KUKA KRL program: MyProgram_045().src

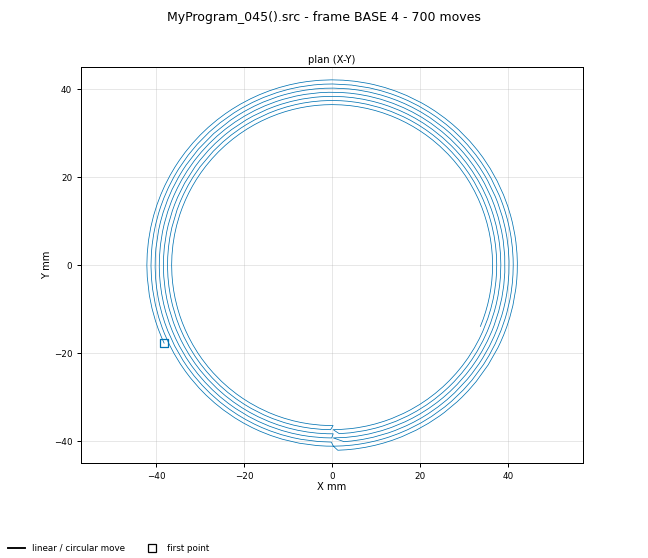
[picture p0: tool path of MyProgram_045().src in frame BASE 4, 700 of 700 moves have a stored position in this frame; points joined in program order, loops and branches not executed]
&ACCESS RVP
&REL 1
&PARAM TEMPLATE = C:\KRC\Roboter\Template\vorgabe
&PARAM EDITMASK = *
DEF MyProgram_045()
; ---- Setting reference (Base) ----
$BASE = BASE_DATA[4]

; --------------------------
; ---- Setting tool (TCP) ----
$TOOL = TOOL_DATA[3]
; --------------------------

$VEL.CP = VEL_APROX_PRINT
Startdeposition()
$VEL.CP = VEL_PRINT
LIN {X -38.1894,Y -17.7476,Z 64,A -162.0836,B 24.8594,C -2.7362,E1 24.8542,E2 -474.5644} C_DIS
LIN {X -38.8026,Y -16.3635,Z 64,A -164.3242,B 24.859,C -2.7399,E1 24.8517,E2 -472.3202} C_DIS
LIN {X -39.5429,Y -14.4833,Z 64,A -167.0478,B 24.8582,C -2.748,E1 24.849,E2 -469.6008} C_DIS
LIN {X -40.1481,Y -12.7091,Z 64,A -169.9379,B 24.8578,C -2.7517,E1 24.8465,E2 -466.703} C_DIS
LIN {X -40.9592,Y -9.7848,Z 64,A -173.7248,B 24.8561,C -2.7677,E1 24.8438,E2 -462.9324} C_DIS
LIN {X -41.5538,Y -6.8335,Z 64,A -178.6112,B 24.8557,C -2.7716,E1 24.8413,E2 -458.0262} C_DIS
LIN {X -42.0235,Y -2.7253,Z 64,A 175.6983,B 24.854,C -2.7884,E1 24.8399,E2 -452.3418} C_DIS
LIN {X -42.113,Y -0.0409,Z 64,A 172.223,B 24.8525,C -2.8017,E1 24.8399,E2 -448.8774} C_DIS
LIN {X -42.0286,Y 2.6491,Z 64,A 168.8043,B 24.8511,C -2.8158,E1 24.8403,E2 -445.4719} C_DIS
LIN {X -41.7458,Y 5.5413,Z 64,A 164.5763,B 24.85,C -2.8253,E1 24.8416,E2 -441.2413} C_DIS
LIN {X -41.2415,Y 8.5177,Z 64,A 160.7229,B 24.8484,C -2.8408,E1 24.8436,E2 -437.4022} C_DIS
LIN {X -40.5761,Y 11.2684,Z 64,A 157.2638,B 24.8467,C -2.8569,E1 24.846,E2 -433.9615} C_DIS
LIN {X -39.798,Y 13.7672,Z 64,A 152.9209,B 24.8464,C -2.8592,E1 24.8498,E2 -429.5994} C_DIS
LIN {X -38.9318,Y 16.0542,Z 64,A 150.3169,B 24.8445,C -2.8771,E1 24.8524,E2 -427.0234} C_DIS
LIN {X -38.035,Y 18.0757,Z 64,A 146.7752,B 24.8442,C -2.88,E1 24.8565,E2 -423.4695} C_DIS
LIN {X -36.8402,Y 20.4016,Z 64,A 143.3193,B 24.8429,C -2.8913,E1 24.8611,E2 -420.0222} C_DIS
LIN {X -35.7285,Y 22.2909,Z 64,A 140.4653,B 24.8419,C -2.901,E1 24.8652,E2 -417.1768} C_DIS
LIN {X -34.7653,Y 23.7657,Z 64,A 138.2662,B 24.8409,C -2.9098,E1 24.8686,E2 -414.9876} C_DIS
LIN {X -33.3953,Y 25.6547,Z 64,A 134.5117,B 24.8407,C -2.9116,E1 24.8749,E2 -411.2193} C_DIS
LIN {X -31.6682,Y 27.7586,Z 64,A 131.0357,B 24.8394,C -2.9235,E1 24.8811,E2 -407.7559} C_DIS
LIN {X -29.9941,Y 29.5595,Z 64,A 127.6294,B 24.8386,C -2.9308,E1 24.8877,E2 -404.3524} C_DIS
LIN {X -28.1817,Y 31.2924,Z 64,A 124.1921,B 24.8378,C -2.9383,E1 24.8947,E2 -400.9189} C_DIS
LIN {X -26.1567,Y 33.0036,Z 64,A 120.4268,B 24.8371,C -2.9441,E1 24.9028,E2 -397.1534} C_DIS
LIN {X -24.2784,Y 34.4092,Z 64,A 117.5539,B 24.836,C -2.9543,E1 24.9093,E2 -394.2946} C_DIS
LIN {X -22.7508,Y 35.4374,Z 64,A 115.1142,B 24.8354,C -2.9598,E1 24.915,E2 -391.8601} C_DIS
LIN {X -20.8416,Y 36.5931,Z 64,A 111.7463,B 24.8352,C -2.9611,E1 24.9231,E2 -388.4851} C_DIS
LIN {X -18.5524,Y 37.8048,Z 64,A 108.1834,B 24.8346,C -2.9662,E1 24.932,E2 -384.925} C_DIS
LIN {X -16.5365,Y 38.7294,Z 64,A 105.4902,B 24.8337,C -2.9746,E1 24.9388,E2 -382.2453} C_DIS
LIN {X -14.2871,Y 39.614,Z 64,A 101.6053,B 24.8341,C -2.9714,E1 24.949,E2 -378.3445} C_DIS
LIN {X -12.0392,Y 40.3542,Z 64,A 98.8345,B 24.833,C -2.9807,E1 24.9563,E2 -375.591} C_DIS
LIN {X -9.7408,Y 40.9696,Z 64,A 95.4963,B 24.8328,C -2.9825,E1 24.9654,E2 -372.2523} C_DIS
LIN {X -7.553,Y 41.4289,Z 64,A 92.4588,B 24.8325,C -2.9849,E1 24.9737,E2 -369.2174} C_DIS
LIN {X -5.5861,Y 41.7398,Z 64,A 89.5891,B 24.8325,C -2.9845,E1 24.9816,E2 -366.3443} C_DIS
LIN {X -2.9978,Y 42.0052,Z 64,A 86.1042,B 24.8323,C -2.9869,E1 24.9913,E2 -362.8635} C_DIS
LIN {X -0.1508,Y 42.1117,Z 64,A 82.6707,B 24.8315,C -2.994,E1 25.0008,E2 -359.4466} C_DIS
LIN {X 2.4941,Y 42.0383,Z 64,A 78.2258,B 24.8328,C -2.9825,E1 25.0133,E2 -354.9755} C_DIS
LIN {X 5.2133,Y 41.7881,Z 64,A 74.8519,B 24.8323,C -2.9867,E1 25.0226,E2 -351.6141} C_DIS
LIN {X 8.0189,Y 41.3412,Z 64,A 71.4094,B 24.8318,C -2.9915,E1 25.0321,E2 -348.1864} C_DIS
LIN {X 9.4728,Y 41.0326,Z 64,A 69.0763,B 24.8324,C -2.986,E1 25.0385,E2 -345.8434} C_DIS
LIN {X 12.0218,Y 40.3594,Z 64,A 65.3773,B 24.8329,C -2.982,E1 25.0484,E2 -342.141} C_DIS
LIN {X 14.4043,Y 39.5717,Z 64,A 62.0211,B 24.8331,C -2.9799,E1 25.0573,E2 -338.7867} C_DIS
LIN {X 16.9832,Y 38.5355,Z 64,A 57.7555,B 24.8344,C -2.9688,E1 25.0683,E2 -334.5046} C_DIS
LIN {X 20.3264,Y 36.882,Z 64,A 53.5076,B 24.8337,C -2.9749,E1 25.0787,E2 -330.2831} C_DIS
LIN {X 21.817,Y 36.0197,Z 64,A 50.7841,B 24.8347,C -2.9657,E1 25.0853,E2 -327.5461} C_DIS
LIN {X 23.4291,Y 34.9933,Z 64,A 48.2049,B 24.8351,C -2.9619,E1 25.0913,E2 -324.9666} C_DIS
LIN {X 25.6673,Y 33.3853,Z 64,A 44.808,B 24.8352,C -2.9611,E1 25.0989,E2 -321.5798} C_DIS
LIN {X 27.3862,Y 31.9908,Z 64,A 41.4445,B 24.8365,C -2.9499,E1 25.1061,E2 -318.2028} C_DIS
LIN {X 28.8143,Y 30.7107,Z 64,A 38.5792,B 24.8375,C -2.9406,E1 25.112,E2 -315.3271} C_DIS
LIN {X 31.3406,Y 28.1278,Z 64,A 34.5739,B 24.837,C -2.9449,E1 25.1197,E2 -311.3493} C_DIS
LIN {X 33.0583,Y 26.0874,Z 64,A 30.6147,B 24.8385,C -2.9312,E1 25.1268,E2 -307.3758} C_DIS
LIN {X 34.283,Y 24.4557,Z 64,A 27.4144,B 24.8401,C -2.9175,E1 25.132,E2 -304.1586} C_DIS
LIN {X 35.9427,Y 21.9439,Z 64,A 23.0552,B 24.8417,C -2.9027,E1 25.1385,E2 -299.7864} C_DIS
LIN {X 37.5319,Y 19.0985,Z 64,A 18.9072,B 24.8425,C -2.8956,E1 25.1439,E2 -295.6435} C_DIS
LIN {X 38.9801,Y 15.9362,Z 64,A 14.6589,B 24.843,C -2.8906,E1 25.1487,E2 -291.4064} C_DIS
LIN {X 39.9208,Y 13.4066,Z 64,A 10.6817,B 24.8447,C -2.8748,E1 25.1524,E2 -287.4142} C_DIS
LIN {X 40.5764,Y 11.2669,Z 64,A 8.1823,B 24.8447,C -2.8751,E1 25.1543,E2 -284.9298} C_DIS
LIN {X 40.9861,Y 9.6717,Z 64,A 5.0679,B 24.847,C -2.8535,E1 25.1564,E2 -281.7822} C_DIS
LIN {X 41.5467,Y 6.8764,Z 64,A 1.8676,B 24.847,C -2.8532,E1 25.158,E2 -278.6001} C_DIS
LIN {X 41.791,Y 5.1908,Z 64,A -0.8122,B 24.8485,C -2.8399,E1 25.1589,E2 -275.9045} C_DIS
LIN {X 42.0276,Y 2.6639,Z 64,A -3.7149,B 24.8486,C -2.8386,E1 25.1596,E2 -273.016} C_DIS
LIN {X 42.1073,Y 0.6196,Z 64,A -6.7943,B 24.8501,C -2.8248,E1 25.1598,E2 -269.9222} C_DIS
LIN {X 42.0818,Y -1.6027,Z 64,A -9.467,B 24.8505,C -2.8213,E1 25.1596,E2 -267.2572} C_DIS
LIN {X 41.9877,Y -3.2337,Z 64,A -11.5891,B 24.851,C -2.8161,E1 25.1592,E2 -265.1353} C_DIS
LIN {X 41.7761,Y -5.3062,Z 64,A -14.9089,B 24.8529,C -2.7988,E1 25.1581,E2 -261.7942} C_DIS
LIN {X 41.0947,Y -9.198,Z 64,A -20.5022,B 24.855,C -2.7783,E1 25.1551,E2 -256.1852} C_DIS
LIN {X 40.3709,Y -11.9829,Z 64,A -23.8222,B 24.8552,C -2.7765,E1 25.1526,E2 -252.8799} C_DIS
LIN {X 39.713,Y -14.0105,Z 64,A -26.748,B 24.8562,C -2.7672,E1 25.15,E2 -249.9486} C_DIS
LIN {X 39.0031,Y -15.8798,Z 64,A -29.3131,B 24.8567,C -2.7617,E1 25.1474,E2 -247.3848} C_DIS
LIN {X 38.2998,Y -17.5081,Z 64,A -31.798,B 24.8576,C -2.7533,E1 25.1446,E2 -244.8936} C_DIS
LIN {X 37.6614,Y -18.8428,Z 64,A -34.6547,B 24.8597,C -2.7331,E1 25.141,E2 -242.0043} C_DIS
LIN {X 35.4698,Y -22.7003,Z 64,A -40.7005,B 24.8615,C -2.7161,E1 25.1322,E2 -235.9491} C_DIS
LIN {X 32.7511,Y -26.4722,Z 64,A -46.2035,B 24.8617,C -2.7132,E1 25.123,E2 -230.4655} C_DIS
LIN {X 30.9506,Y -28.5566,Z 64,A -49.7785,B 24.8624,C -2.7067,E1 25.1164,E2 -226.8911} C_DIS
LIN {X 29.5084,Y -30.0446,Z 64,A -52.2115,B 24.8624,C -2.7064,E1 25.1116,E2 -224.4677} C_DIS
LIN {X 28.4019,Y -31.0925,Z 64,A -55.2369,B 24.8645,C -2.686,E1 25.1053,E2 -221.4062} C_DIS
LIN {X 25.523,Y -33.4965,Z 64,A -59.4397,B 24.8641,C -2.6897,E1 25.0963,E2 -217.2281} C_DIS
LIN {X 24.4241,Y -34.3055,Z 64,A -61.7378,B 24.8652,C -2.6788,E1 25.091,E2 -214.9122} C_DIS
LIN {X 21.9075,Y -35.9646,Z 64,A -65.825,B 24.866,C -2.6713,E1 25.0814,E2 -210.8205} C_DIS
LIN {X 19.1281,Y -37.5169,Z 64,A -70.6189,B 24.8675,C -2.6567,E1 25.0695,E2 -206.0057} C_DIS
LIN {X 15.8604,Y -39.0109,Z 64,A -74.9095,B 24.8672,C -2.6589,E1 25.0586,E2 -201.7306} C_DIS
LIN {X 13.743,Y -39.8058,Z 64,A -77.6711,B 24.8672,C -2.6598,E1 25.0514,E2 -198.977} C_DIS
LIN {X 11.7789,Y -40.4308,Z 64,A -80.9256,B 24.8682,C -2.6497,E1 25.0426,E2 -195.7043} C_DIS
LIN {X 9.793,Y -40.9572,Z 64,A -83.3321,B 24.8678,C -2.6529,E1 25.0362,E2 -193.3089} C_DIS
LIN {X 7.5807,Y -41.4241,Z 64,A -87.0071,B 24.869,C -2.6413,E1 25.026,E2 -189.6109} C_DIS
LIN {X 5.2253,Y -41.7866,Z 64,A -89.7045,B 24.8684,C -2.6473,E1 25.0186,E2 -186.9299} C_DIS
LIN {X 3.3156,Y -41.9811,Z 64,A -92.4426,B 24.8687,C -2.6441,E1 25.011,E2 -184.1858} C_DIS
LIN {X 1.2963,Y -42.0919,Z 64,A -95.1766,B 24.8688,C -2.6433,E1 25.0034,E2 -181.4508} C_DIS
LIN {X 1.2963,Y -42.0919,Z 64,A -95.1766,B 24.8688,C -2.6433,E1 25.0034,E2 -181.4508} C_DIS
Enddeposition()
LIN {X 0.2865,Y -41.1698,Z 64,A -95.4325,B 24.8656,C -2.6754,E1 25.0029,E2 -181.2711} C_DIS
Startdeposition()
$VEL.CP = VEL_PRINT
LIN {X 2.5086,Y -41.0971,Z 64,A -91.9997,B 24.865,C -2.6814,E1 25.0125,E2 -184.7172} C_DIS
LIN {X 4.5975,Y -40.9157,Z 64,A -89.3544,B 24.8652,C -2.679,E1 25.0198,E2 -187.3551} C_DIS
LIN {X 6.285,Y -40.6906,Z 64,A -86.9492,B 24.865,C -2.6811,E1 25.0264,E2 -189.7631} C_DIS
LIN {X 7.9842,Y -40.3918,Z 64,A -84.5187,B 24.8648,C -2.6835,E1 25.0331,E2 -192.1965} C_DIS
LIN {X 9.725,Y -40.0081,Z 64,A -81.9886,B 24.8645,C -2.6865,E1 25.04,E2 -194.7304} C_DIS
LIN {X 11.6702,Y -39.4844,Z 64,A -79.4566,B 24.8645,C -2.6854,E1 25.0468,E2 -197.2555} C_DIS
LIN {X 12.9333,Y -39.0895,Z 64,A -77.251,B 24.8638,C -2.6932,E1 25.0527,E2 -199.4754} C_DIS
LIN {X 15.0733,Y -38.3145,Z 64,A -74.3091,B 24.8638,C -2.6939,E1 25.0604,E2 -202.4126} C_DIS
LIN {X 17.1775,Y -37.4189,Z 64,A -70.4429,B 24.8621,C -2.7094,E1 25.0703,E2 -206.3061} C_DIS
LIN {X 20.208,Y -35.8732,Z 64,A -66.3938,B 24.8624,C -2.7063,E1 25.0802,E2 -210.3366} C_DIS
LIN {X 22.5789,Y -34.43,Z 64,A -61.6674,B 24.8603,C -2.7275,E1 25.0915,E2 -215.098} C_DIS
LIN {X 25.5833,Y -32.2598,Z 64,A -57.4368,B 24.8607,C -2.723,E1 25.1008,E2 -219.3026} C_DIS
LIN {X 27.1419,Y -30.9604,Z 64,A -54.1094,B 24.8592,C -2.7376,E1 25.1079,E2 -222.6515} C_DIS
LIN {X 29.8248,Y -28.3855,Z 64,A -48.7405,B 24.8576,C -2.7531,E1 25.1185,E2 -228.0344} C_DIS
LIN {X 31.799,Y -26.1552,Z 64,A -44.4279,B 24.8562,C -2.7665,E1 25.1263,E2 -232.359} C_DIS
LIN {X 34.4182,Y -22.5969,Z 64,A -39.348,B 24.8564,C -2.7649,E1 25.1344,E2 -237.4102} C_DIS
LIN {X 35.7205,Y -20.4761,Z 64,A -35.0283,B 24.8539,C -2.7892,E1 25.1406,E2 -241.7654} C_DIS
LIN {X 37.076,Y -17.9054,Z 64,A -31.2501,B 24.8531,C -2.7964,E1 25.1453,E2 -245.5404} C_DIS
LIN {X 38.4017,Y -14.8515,Z 64,A -26.6876,B 24.8518,C -2.809,E1 25.1502,E2 -250.1076} C_DIS
LIN {X 39.3357,Y -12.1622,Z 64,A -23.3798,B 24.8517,C -2.8098,E1 25.1531,E2 -253.3986} C_DIS
LIN {X 39.709,Y -10.8824,Z 64,A -21.0005,B 24.8501,C -2.8246,E1 25.1549,E2 -255.7991} C_DIS
LIN {X 40.3965,Y -7.9597,Z 64,A -17.258,B 24.8495,C -2.83,E1 25.1571,E2 -259.5328} C_DIS
LIN {X 40.6939,Y -6.2639,Z 64,A -14.7095,B 24.8485,C -2.8401,E1 25.1582,E2 -262.0904} C_DIS
LIN {X 40.9627,Y -4.1566,Z 64,A -11.8666,B 24.8477,C -2.8475,E1 25.1591,E2 -264.9337} C_DIS
LIN {X 41.1159,Y -2.1722,Z 64,A -9.0364,B 24.8466,C -2.8572,E1 25.1597,E2 -267.7702} C_DIS
LIN {X 41.1733,Y 0.0875,Z 64,A -6.0721,B 24.8459,C -2.864,E1 25.1597,E2 -270.7328} C_DIS
LIN {X 41.1424,Y 1.5996,Z 64,A -3.8198,B 24.8449,C -2.8731,E1 25.1596,E2 -272.9934} C_DIS
LIN {X 40.9794,Y 3.9883,Z 64,A -0.3005,B 24.8434,C -2.8867,E1 25.1587,E2 -276.5239} C_DIS
LIN {X 40.6864,Y 6.3124,Z 64,A 2.5108,B 24.8432,C -2.889,E1 25.1576,E2 -279.3241} C_DIS
LIN {X 40.3371,Y 8.2546,Z 64,A 5.8381,B 24.8412,C -2.9073,E1 25.1559,E2 -282.6755} C_DIS
LIN {X 39.8463,Y 10.3687,Z 64,A 8.2951,B 24.8412,C -2.9067,E1 25.1542,E2 -285.1167} C_DIS
LIN {X 39.3395,Y 12.1503,Z 64,A 10.9164,B 24.8403,C -2.915,E1 25.1521,E2 -287.7428} C_DIS
LIN {X 38.7443,Y 13.9319,Z 64,A 13.5664,B 24.8394,C -2.9232,E1 25.1497,E2 -290.3973} C_DIS
LIN {X 38.0364,Y 15.7633,Z 64,A 17.5379,B 24.8362,C -2.9521,E1 25.1454,E2 -294.4152} C_DIS
LIN {X 36.1894,Y 19.6355,Z 64,A 22.4347,B 24.8365,C -2.9499,E1 25.1392,E2 -299.2809} C_DIS
LIN {X 35.0453,Y 21.6121,Z 64,A 25.3732,B 24.836,C -2.9541,E1 25.135,E2 -302.2144} C_DIS
LIN {X 33.9192,Y 23.339,Z 64,A 28.1541,B 24.8354,C -2.9598,E1 25.1307,E2 -304.995} C_DIS
LIN {X 32.6665,Y 25.0626,Z 64,A 31.3409,B 24.8342,C -2.9706,E1 25.1253,E2 -308.192} C_DIS
LIN {X 30.7767,Y 27.3504,Z 64,A 35.0878,B 24.8338,C -2.9737,E1 25.1186,E2 -311.9291} C_DIS
LIN {X 29.3498,Y 28.876,Z 64,A 38.5961,B 24.832,C -2.9896,E1 25.1118,E2 -315.46} C_DIS
LIN {X 27.6483,Y 30.51,Z 64,A 41.6362,B 24.8317,C -2.9921,E1 25.1055,E2 -318.4938} C_DIS
LIN {X 25.9223,Y 31.9884,Z 64,A 44.7794,B 24.8311,C -2.9977,E1 25.0988,E2 -321.6382} C_DIS
LIN {X 23.7335,Y 33.6442,Z 64,A 48.6249,B 24.8303,C -3.0045,E1 25.0901,E2 -325.4862} C_DIS
LIN {X 22.074,Y 34.7558,Z 64,A 51.5102,B 24.8297,C -3.0105,E1 25.0833,E2 -328.3762} C_DIS
LIN {X 19.6272,Y 36.1939,Z 64,A 55.2494,B 24.8294,C -3.0126,E1 25.0742,E2 -332.1095} C_DIS
LIN {X 17.2767,Y 37.3731,Z 64,A 58.8016,B 24.8291,C -3.0153,E1 25.0653,E2 -335.6587} C_DIS
LIN {X 15.2195,Y 38.2569,Z 64,A 61.8902,B 24.8288,C -3.0181,E1 25.0574,E2 -338.7467} C_DIS
LIN {X 13.3989,Y 38.9323,Z 64,A 64.4426,B 24.8288,C -3.0181,E1 25.0507,E2 -341.2942} C_DIS
LIN {X 11.048,Y 39.6629,Z 64,A 68.5273,B 24.8274,C -3.0303,E1 25.0397,E2 -345.4006} C_DIS
LIN {X 8.5196,Y 40.2823,Z 64,A 72.2473,B 24.827,C -3.0334,E1 25.0295,E2 -349.1232} C_DIS
LIN {X 4.4101,Y 40.9362,Z 64,A 78.0835,B 24.8268,C -3.0354,E1 25.0134,E2 -354.9592} C_DIS
LIN {X 0.0841,Y 41.1734,Z 64,A 83.1585,B 24.8284,C -3.0216,E1 24.9993,E2 -359.9999} C_DIS
LIN {X -1.8757,Y 41.1298,Z 64,A 86.0866,B 24.8282,C -3.0235,E1 24.9911,E2 -362.9331} C_DIS
LIN {X -4.1334,Y 40.9648,Z 64,A 89.7492,B 24.8275,C -3.029,E1 24.9809,E2 -366.6105} C_DIS
LIN {X -7.42,Y 40.4984,Z 64,A 94.0771,B 24.8284,C -3.0219,E1 24.969,E2 -370.9255} C_DIS
LIN {X -9.8107,Y 39.9866,Z 64,A 97.8152,B 24.8282,C -3.0232,E1 24.9588,E2 -374.6717} C_DIS
LIN {X -12.5005,Y 39.2294,Z 64,A 101.6871,B 24.8287,C -3.0188,E1 24.9485,E2 -378.5396} C_DIS
LIN {X -15.6079,Y 38.1002,Z 64,A 105.9096,B 24.8299,C -3.008,E1 24.9375,E2 -382.7452} C_DIS
LIN {X -18.1335,Y 36.9647,Z 64,A 110.0885,B 24.8301,C -3.0062,E1 24.9269,E2 -386.9305} C_DIS
LIN {X -20.4211,Y 35.7522,Z 64,A 113.368,B 24.8313,C -2.9962,E1 24.9189,E2 -390.1954} C_DIS
LIN {X -22.2692,Y 34.6311,Z 64,A 116.6839,B 24.8315,C -2.9944,E1 24.9111,E2 -393.5176} C_DIS
LIN {X -25.4707,Y 32.3492,Z 64,A 122.5841,B 24.8321,C -2.9884,E1 24.8979,E2 -399.4246} C_DIS
LIN {X -27.954,Y 30.2292,Z 64,A 127.0418,B 24.8334,C -2.9773,E1 24.8886,E2 -403.8734} C_DIS
LIN {X -30.6733,Y 27.4659,Z 64,A 131.8749,B 24.8356,C -2.9577,E1 24.8794,E2 -408.6808} C_DIS
LIN {X -32.7326,Y 24.976,Z 64,A 137.3602,B 24.8356,C -2.9575,E1 24.8699,E2 -414.1913} C_DIS
LIN {X -34.9355,Y 21.7886,Z 64,A 141.9022,B 24.8383,C -2.9332,E1 24.8629,E2 -418.6978} C_DIS
LIN {X -36.0094,Y 19.964,Z 64,A 144.704,B 24.8394,C -2.9232,E1 24.8591,E2 -421.4905} C_DIS
LIN {X -37.206,Y 17.6331,Z 64,A 149.0173,B 24.8398,C -2.9201,E1 24.8537,E2 -425.8195} C_DIS
LIN {X -38.2384,Y 15.2655,Z 64,A 152.1055,B 24.8416,C -2.9038,E1 24.8505,E2 -428.886} C_DIS
LIN {X -38.9655,Y 13.3009,Z 64,A 154.8405,B 24.8427,C -2.8931,E1 24.8479,E2 -431.6108} C_DIS
LIN {X -39.4625,Y 11.7441,Z 64,A 157.4607,B 24.8431,C -2.8899,E1 24.8458,E2 -434.2385} C_DIS
LIN {X -40.1258,Y 9.226,Z 64,A 160.9334,B 24.8445,C -2.8771,E1 24.8434,E2 -437.7007} C_DIS
LIN {X -40.5485,Y 7.1441,Z 64,A 164.202,B 24.8451,C -2.8712,E1 24.8417,E2 -440.9748} C_DIS
LIN {X -40.908,Y 4.6637,Z 64,A 167.3897,B 24.8466,C -2.8571,E1 24.8406,E2 -444.1476} C_DIS
LIN {X -41.0794,Y 2.777,Z 64,A 170.5921,B 24.8469,C -2.8549,E1 24.8399,E2 -447.3641} C_DIS
LIN {X -41.1735,Y -0.1582,Z 64,A 174.2183,B 24.8488,C -2.8371,E1 24.8399,E2 -450.9696} C_DIS
LIN {X -41.0704,Y -2.9085,Z 64,A 178.4713,B 24.8496,C -2.8298,E1 24.8404,E2 -455.2307} C_DIS
LIN {X -40.8091,Y -5.4637,Z 64,A -177.2907,B 24.85,C -2.8261,E1 24.842,E2 -459.4852} C_DIS
LIN {X -40.1744,Y -9.0147,Z 64,A -172.6624,B 24.852,C -2.8066,E1 24.8446,E2 -464.0939} C_DIS
LIN {X -39.3951,Y -11.968,Z 64,A -168.8506,B 24.8539,C -2.7891,E1 24.8475,E2 -467.8861} C_DIS
LIN {X -38.6067,Y -14.3098,Z 64,A -165.727,B 24.8553,C -2.7757,E1 24.8503,E2 -470.9953} C_DIS
LIN {X -38.0815,Y -15.6538,Z 64,A -163.3316,B 24.8554,C -2.7744,E1 24.8529,E2 -473.4009} C_DIS
LIN {X -37.0242,Y -18.0118,Z 64,A -159.7863,B 24.8565,C -2.7639,E1 24.857,E2 -476.9406} C_DIS
LIN {X -35.9413,Y -20.0861,Z 64,A -156.5193,B 24.8574,C -2.7554,E1 24.8614,E2 -480.2044} C_DIS
LIN {X -34.5038,Y -22.4664,Z 64,A -153.0233,B 24.8589,C -2.7412,E1 24.8665,E2 -483.6844} C_DIS
LIN {X -33.3226,Y -24.1831,Z 64,A -149.6937,B 24.8591,C -2.7392,E1 24.8719,E2 -487.0255} C_DIS
LIN {X -32.1984,Y -25.6616,Z 64,A -147.4173,B 24.8601,C -2.7295,E1 24.8758,E2 -489.2896} C_DIS
LIN {X -30.2484,Y -27.9335,Z 64,A -142.9089,B 24.8606,C -2.7244,E1 24.8841,E2 -493.8059} C_DIS
LIN {X -28.677,Y -29.5441,Z 64,A -139.7292,B 24.8612,C -2.7185,E1 24.8904,E2 -496.9851} C_DIS
LIN {X -26.7059,Y -31.3372,Z 64,A -135.5112,B 24.8612,C -2.7177,E1 24.8993,E2 -501.2178} C_DIS
LIN {X -24.7341,Y -32.9158,Z 64,A -132.1941,B 24.8622,C -2.7092,E1 24.9066,E2 -504.5265} C_DIS
LIN {X -22.1397,Y -34.7142,Z 64,A -128.359,B 24.8636,C -2.6953,E1 24.9155,E2 -508.3413} C_DIS
LIN {X -20.1713,Y -35.8937,Z 64,A -124.7588,B 24.8635,C -2.6961,E1 24.9242,E2 -511.9541} C_DIS
LIN {X -18.1009,Y -36.9807,Z 64,A -121.751,B 24.8642,C -2.689,E1 24.9316,E2 -514.953} C_DIS
LIN {X -16.336,Y -37.7938,Z 64,A -119.1423,B 24.8646,C -2.6848,E1 24.9383,E2 -517.558} C_DIS
LIN {X -13.9314,Y -38.7442,Z 64,A -114.6456,B 24.8637,C -2.6936,E1 24.9501,E2 -522.085} C_DIS
LIN {X -11.2823,Y -39.5972,Z 64,A -111.0518,B 24.8644,C -2.6872,E1 24.9597,E2 -525.6695} C_DIS
LIN {X -7.4714,Y -40.49,Z 64,A -105.4146,B 24.8644,C -2.6875,E1 24.9751,E2 -531.3141} C_DIS
LIN {X -3.4297,Y -41.0302,Z 64,A -100.7188,B 24.8658,C -2.6729,E1 24.9881,E2 -535.9783} C_DIS
LIN {X -1.2919,Y -41.1526,Z 64,A -97.2547,B 24.8651,C -2.6801,E1 24.9978,E2 -539.4603} C_DIS
LIN {X 0.2865,Y -41.1698,Z 64,A -95.4322,B 24.8656,C -2.6752,E1 25.0028,E2 -541.2711} C_DIS
Enddeposition()
LIN {X 0.2865,Y -41.1698,Z 64,A -95.4322,B 24.8656,C -2.6752,E1 25.0028,E2 -541.2711} C_DIS
Startdeposition()
$VEL.CP = VEL_PRINT
LIN {X -0.1805,Y -40.2341,Z 64,A -98.0882,B 24.8668,C -2.6637,E1 24.9954,E2 -538.5877} C_DIS
LIN {X -3.0801,Y -40.1166,Z 64,A -102.2428,B 24.8668,C -2.6633,E1 24.9838,E2 -534.4307} C_DIS
LIN {X -7.069,Y -39.6085,Z 64,A -106.6261,B 24.8649,C -2.6824,E1 24.9718,E2 -530.0892} C_DIS
LIN {X -8.9428,Y -39.228,Z 64,A -110.237,B 24.8659,C -2.6719,E1 24.9618,E2 -526.449} C_DIS
LIN {X -11.5498,Y -38.5411,Z 64,A -114.2477,B 24.8659,C -2.6722,E1 24.9511,E2 -522.4326} C_DIS
LIN {X -14.0314,Y -37.7088,Z 64,A -117.4029,B 24.8649,C -2.6825,E1 24.9428,E2 -519.2958} C_DIS
LIN {X -15.8936,Y -36.9625,Z 64,A -120.4809,B 24.8649,C -2.6825,E1 24.9348,E2 -516.2109} C_DIS
LIN {X -17.6351,Y -36.1637,Z 64,A -122.897,B 24.8642,C -2.6895,E1 24.9288,E2 -513.8053} C_DIS
LIN {X -19.656,Y -35.1063,Z 64,A -126.8213,B 24.8646,C -2.6855,E1 24.9191,E2 -509.8603} C_DIS
LIN {X -21.4529,Y -34.0383,Z 64,A -129.7071,B 24.864,C -2.691,E1 24.9123,E2 -506.9785} C_DIS
LIN {X -23.5252,Y -32.6407,Z 64,A -133.0557,B 24.8632,C -2.6992,E1 24.9046,E2 -503.6381} C_DIS
LIN {X -25.4872,Y -31.1328,Z 64,A -137.2174,B 24.8632,C -2.6981,E1 24.8955,E2 -499.4583} C_DIS
LIN {X -27.7086,Y -29.1733,Z 64,A -140.5996,B 24.8615,C -2.7159,E1 24.8886,E2 -496.1048} C_DIS
LIN {X -29.5736,Y -27.2804,Z 64,A -145.098,B 24.8615,C -2.7159,E1 24.8799,E2 -491.5869} C_DIS
LIN {X -31.387,Y -25.1736,Z 64,A -148.404,B 24.8598,C -2.7321,E1 24.874,E2 -488.3043} C_DIS
LIN {X -32.8459,Y -23.2376,Z 64,A -151.6868,B 24.8588,C -2.7422,E1 24.8686,E2 -485.0299} C_DIS
LIN {X -33.9156,Y -21.6461,Z 64,A -155.2793,B 24.859,C -2.7397,E1 24.8631,E2 -481.4133} C_DIS
LIN {X -35.7912,Y -18.3795,Z 64,A -160.7908,B 24.8577,C -2.7524,E1 24.8558,E2 -475.903} C_DIS
LIN {X -37.3572,Y -14.9411,Z 64,A -165.3717,B 24.8553,C -2.7758,E1 24.8507,E2 -471.3528} C_DIS
LIN {X -38.0454,Y -13.0913,Z 64,A -168.4206,B 24.8547,C -2.7814,E1 24.8478,E2 -468.2999} C_DIS
LIN {X -38.6307,Y -11.2458,Z 64,A -171.1999,B 24.8539,C -2.7892,E1 24.8456,E2 -465.5235} C_DIS
LIN {X -39.238,Y -8.8999,Z 64,A -174.1639,B 24.8522,C -2.8046,E1 24.8436,E2 -462.5789} C_DIS
LIN {X -39.5518,Y -7.3813,Z 64,A -177.0935,B 24.8523,C -2.8038,E1 24.842,E2 -459.6302} C_DIS
LIN {X -39.9087,Y -5.1097,Z 64,A -179.9512,B 24.8508,C -2.8182,E1 24.8409,E2 -456.7897} C_DIS
LIN {X -40.1125,Y -3.1313,Z 64,A 176.7016,B 24.8504,C -2.8217,E1 24.8401,E2 -453.4309} C_DIS
LIN {X -40.2305,Y -0.5686,Z 64,A 173.3305,B 24.8489,C -2.836,E1 24.8398,E2 -450.0737} C_DIS
LIN {X -40.1994,Y 1.6805,Z 64,A 170.003,B 24.848,C -2.8447,E1 24.84,E2 -446.7472} C_DIS
LIN {X -40.0572,Y 3.7726,Z 64,A 166.3891,B 24.8476,C -2.8478,E1 24.8409,E2 -443.1189} C_DIS
LIN {X -39.4504,Y 7.9051,Z 64,A 161.238,B 24.8448,C -2.8744,E1 24.8433,E2 -438.0008} C_DIS
LIN {X -39.0144,Y 9.8343,Z 64,A 157.9698,B 24.8443,C -2.8785,E1 24.8454,E2 -434.7233} C_DIS
LIN {X -38.4229,Y 11.9365,Z 64,A 154.882,B 24.8433,C -2.8883,E1 24.8479,E2 -431.6411} C_DIS
LIN {X -37.3996,Y 14.835,Z 64,A 151.2634,B 24.841,C -2.9092,E1 24.8513,E2 -428.0521} C_DIS
LIN {X -36.3732,Y 17.1986,Z 64,A 146.37,B 24.8412,C -2.9074,E1 24.857,E2 -423.1275} C_DIS
LIN {X -34.8808,Y 20.0534,Z 64,A 142.5299,B 24.8389,C -2.9282,E1 24.8621,E2 -419.3169} C_DIS
LIN {X -33.9616,Y 21.5734,Z 64,A 140.0794,B 24.838,C -2.936,E1 24.8656,E2 -416.8726} C_DIS
LIN {X -33.1653,Y 22.7792,Z 64,A 137.0638,B 24.8385,C -2.9315,E1 24.8704,E2 -413.8313} C_DIS
LIN {X -30.3883,Y 26.37,Z 64,A 130.2426,B 24.8371,C -2.9442,E1 24.8825,E2 -407.0089} C_DIS
LIN {X -26.9047,Y 29.9158,Z 64,A 123.127,B 24.8353,C -2.9602,E1 24.8969,E2 -399.9021} C_DIS
LIN {X -23.1721,Y 32.892,Z 64,A 117.3757,B 24.8325,C -2.9858,E1 24.9095,E2 -394.191} C_DIS
LIN {X -21.483,Y 34.0193,Z 64,A 114.4692,B 24.8319,C -2.991,E1 24.9163,E2 -391.2876} C_DIS
LIN {X -19.9857,Y 34.9197,Z 64,A 112.1765,B 24.8311,C -2.9976,E1 24.9218,E2 -389.0038} C_DIS
LIN {X -17.7145,Y 36.1247,Z 64,A 107.5857,B 24.8317,C -2.9927,E1 24.9333,E2 -384.3888} C_DIS
LIN {X -15.6604,Y 37.0616,Z 64,A 104.5516,B 24.8309,C -2.9993,E1 24.9411,E2 -381.3634} C_DIS
LIN {X -12.3091,Y 38.3054,Z 64,A 100.4025,B 24.8289,C -3.0169,E1 24.9519,E2 -377.2482} C_DIS
LIN {X -10.7876,Y 38.7611,Z 64,A 97.3706,B 24.8297,C -3.0099,E1 24.9601,E2 -374.1946} C_DIS
LIN {X -8.4549,Y 39.3362,Z 64,A 94.2275,B 24.829,C -3.0163,E1 24.9686,E2 -371.0628} C_DIS
LIN {X -6.1572,Y 39.7605,Z 64,A 90.5754,B 24.8292,C -3.0146,E1 24.9787,E2 -367.4032} C_DIS
LIN {X -3.8372,Y 40.051,Z 64,A 87.7531,B 24.8282,C -3.0229,E1 24.9865,E2 -364.5987} C_DIS
LIN {X -1.6497,Y 40.2007,Z 64,A 84.6564,B 24.8281,C -3.0244,E1 24.9951,E2 -361.5046} C_DIS
LIN {X 0.3608,Y 40.233,Z 64,A 80.9768,B 24.8292,C -3.0143,E1 25.0054,E2 -357.8011} C_DIS
LIN {X 3.8068,Y 40.0537,Z 64,A 76.7063,B 24.8283,C -3.0227,E1 25.0173,E2 -353.5526} C_DIS
LIN {X 5.9003,Y 39.7994,Z 64,A 73.4227,B 24.8288,C -3.0182,E1 25.0264,E2 -350.2612} C_DIS
LIN {X 8.4806,Y 39.3306,Z 64,A 69.3609,B 24.8295,C -3.0122,E1 25.0375,E2 -346.1899} C_DIS
LIN {X 11.0934,Y 38.6749,Z 64,A 66.2504,B 24.8286,C -3.0199,E1 25.0458,E2 -343.1026} C_DIS
LIN {X 12.9494,Y 38.0937,Z 64,A 63.2769,B 24.8292,C -3.0148,E1 25.0538,E2 -340.1227} C_DIS
LIN {X 14.7788,Y 37.4219,Z 64,A 60.7117,B 24.8292,C -3.0152,E1 25.0604,E2 -337.564} C_DIS
LIN {X 16.5281,Y 36.6828,Z 64,A 57.837,B 24.8297,C -3.0099,E1 25.0678,E2 -334.6836} C_DIS
LIN {X 18.2374,Y 35.8635,Z 64,A 55.4014,B 24.8297,C -3.0104,E1 25.0739,E2 -332.2559} C_DIS
LIN {X 20.2009,Y 34.7958,Z 64,A 51.5765,B 24.8312,C -2.9967,E1 25.0832,E2 -328.4095} C_DIS
LIN {X 22.2003,Y 33.5553,Z 64,A 47.8681,B 24.8324,C -2.9862,E1 25.0919,E2 -324.6885} C_DIS
LIN {X 25.4347,Y 31.1753,Z 64,A 43.0963,B 24.8319,C -2.9905,E1 25.1025,E2 -319.9443} C_DIS
LIN {X 26.8184,Y 29.9931,Z 64,A 40.5081,B 24.8325,C -2.9856,E1 25.1079,E2 -317.3546} C_DIS
LIN {X 28.5167,Y 28.3836,Z 64,A 37.033,B 24.8335,C -2.9766,E1 25.1149,E2 -313.8726} C_DIS
LIN {X 30.1104,Y 26.6873,Z 64,A 33.4543,B 24.8348,C -2.9652,E1 25.1216,E2 -310.2829} C_DIS
LIN {X 32.0978,Y 24.26,Z 64,A 29.66,B 24.8348,C -2.9654,E1 25.1282,E2 -306.5068} C_DIS
LIN {X 33.5299,Y 22.2387,Z 64,A 25.4715,B 24.8369,C -2.9463,E1 25.1349,E2 -302.2935} C_DIS
LIN {X 34.6875,Y 20.3862,Z 64,A 22.8825,B 24.8369,C -2.9466,E1 25.1386,E2 -299.7185} C_DIS
LIN {X 35.3611,Y 19.1937,Z 64,A 20.3578,B 24.8384,C -2.9322,E1 25.142,E2 -297.1729} C_DIS
LIN {X 37.0912,Y 15.5901,Z 64,A 15.2212,B 24.8392,C -2.9255,E1 25.148,E2 -292.0482} C_DIS
LIN {X 37.6471,Y 14.1954,Z 64,A 12.5741,B 24.8408,C -2.9111,E1 25.1507,E2 -289.3818} C_DIS
LIN {X 38.737,Y 10.8736,Z 64,A 7.9772,B 24.8417,C -2.9027,E1 25.1544,E2 -284.7912} C_DIS
LIN {X 39.3247,Y 8.5075,Z 64,A 4.5918,B 24.8427,C -2.8937,E1 25.1566,E2 -281.4041} C_DIS
LIN {X 39.738,Y 6.3031,Z 64,A 1.6451,B 24.8433,C -2.888,E1 25.158,E2 -278.4613} C_DIS
LIN {X 40.0609,Y 3.7329,Z 64,A -2.863,B 24.846,C -2.8631,E1 25.1594,E2 -273.9208} C_DIS
LIN {X 40.2239,Y 0.9243,Z 64,A -6.5556,B 24.8468,C -2.8558,E1 25.1598,E2 -270.2328} C_DIS
LIN {X 40.1897,Y -1.8946,Z 64,A -10.2738,B 24.8476,C -2.8481,E1 25.1595,E2 -266.5185} C_DIS
LIN {X 39.9994,Y -4.3418,Z 64,A -13.7534,B 24.8488,C -2.8374,E1 25.1586,E2 -263.0342} C_DIS
LIN {X 39.717,Y -6.435,Z 64,A -16.5413,B 24.8494,C -2.8316,E1 25.1575,E2 -260.249} C_DIS
LIN {X 39.3873,Y -8.2138,Z 64,A -19.1906,B 24.8504,C -2.8223,E1 25.156,E2 -257.5933} C_DIS
LIN {X 39.0029,Y -9.8788,Z 64,A -21.505,B 24.851,C -2.8168,E1 25.1545,E2 -255.2792} C_DIS
LIN {X 38.5982,Y -11.3569,Z 64,A -24.1511,B 24.8525,C -2.8024,E1 25.1524,E2 -252.6141} C_DIS
LIN {X 37.6029,Y -14.3121,Z 64,A -27.9671,B 24.8528,C -2.7992,E1 25.1489,E2 -248.8122} C_DIS
LIN {X 36.8833,Y -16.0759,Z 64,A -31.1581,B 24.8545,C -2.7833,E1 25.1454,E2 -245.6009} C_DIS
LIN {X 35.7401,Y -18.4794,Z 64,A -35.1912,B 24.8561,C -2.7683,E1 25.1404,E2 -241.5538} C_DIS
LIN {X 34.1979,Y -21.1971,Z 64,A -38.8663,B 24.8561,C -2.7684,E1 25.1352,E2 -237.898} C_DIS
LIN {X 33.4089,Y -22.4205,Z 64,A -41.2922,B 24.8572,C -2.757,E1 25.1314,E2 -235.4571} C_DIS
LIN {X 31.7874,Y -24.6656,Z 64,A -44.6875,B 24.8574,C -2.7554,E1 25.1258,E2 -232.0744} C_DIS
LIN {X 30.7545,Y -25.9423,Z 64,A -48.2665,B 24.8601,C -2.7296,E1 25.1193,E2 -228.4505} C_DIS
LIN {X 27.862,Y -29.0262,Z 64,A -53.2831,B 24.8599,C -2.7311,E1 25.1096,E2 -223.4589} C_DIS
LIN {X 26.1675,Y -30.5627,Z 64,A -56.9799,B 24.8614,C -2.7168,E1 25.1018,E2 -219.7431} C_DIS
LIN {X 24.1252,Y -32.1992,Z 64,A -60.4321,B 24.8617,C -2.7133,E1 25.0942,E2 -216.2952} C_DIS
LIN {X 21.8544,Y -33.7816,Z 64,A -64.2852,B 24.8624,C -2.707,E1 25.0853,E2 -212.4402} C_DIS
LIN {X 20.2747,Y -34.7534,Z 64,A -66.7457,B 24.8626,C -2.705,E1 25.0794,E2 -209.9825} C_DIS
LIN {X 18.5684,Y -35.6934,Z 64,A -69.9131,B 24.8637,C -2.6944,E1 25.0715,E2 -206.7989} C_DIS
LIN {X 16.9095,Y -36.5087,Z 64,A -72.6994,B 24.8643,C -2.688,E1 25.0645,E2 -204.0047} C_DIS
LIN {X 14.2819,Y -37.6143,Z 64,A -76.1807,B 24.864,C -2.691,E1 25.0555,E2 -200.5384} C_DIS
LIN {X 12.7612,Y -38.1572,Z 64,A -79.0565,B 24.8652,C -2.6797,E1 25.0478,E2 -197.6413} C_DIS
LIN {X 9.3709,Y -39.1277,Z 64,A -83.6127,B 24.865,C -2.6813,E1 25.0356,E2 -193.0961} C_DIS
LIN {X 6.8812,Y -39.6413,Z 64,A -87.3762,B 24.8655,C -2.6763,E1 25.0252,E2 -189.3252} C_DIS
LIN {X 4.4242,Y -39.9901,Z 64,A -91.0207,B 24.8659,C -2.6725,E1 25.0151,E2 -185.6747} C_DIS
LIN {X 2.7156,Y -40.1427,Z 64,A -94.0689,B 24.8668,C -2.6631,E1 25.0066,E2 -182.6053} C_DIS
LIN {X 2.7156,Y -40.1427,Z 64,A -94.0689,B 24.8668,C -2.6631,E1 25.0066,E2 -182.6053} C_DIS
Enddeposition()
LIN {X 0.2668,Y -39.2896,Z 64,A -95.3819,B 24.8623,C -2.7083,E1 25.0032,E2 -181.4001} C_DIS
Startdeposition()
$VEL.CP = VEL_PRINT
LIN {X 3.0992,Y -39.1733,Z 64,A -90.7175,B 24.8613,C -2.7173,E1 25.0163,E2 -186.0841} C_DIS
LIN {X 5.7436,Y -38.8741,Z 64,A -87.1996,B 24.8616,C -2.7146,E1 25.026,E2 -189.5927} C_DIS
LIN {X 8.3849,Y -38.3907,Z 64,A -83.2697,B 24.8612,C -2.7181,E1 25.0367,E2 -193.5261} C_DIS
LIN {X 11.2922,Y -37.6381,Z 64,A -78.7724,B 24.8606,C -2.7244,E1 25.0489,E2 -198.0312} C_DIS
LIN {X 13.4851,Y -36.9093,Z 64,A -75.2628,B 24.8599,C -2.7308,E1 25.0581,E2 -201.5487} C_DIS
LIN {X 16.5987,Y -35.6179,Z 64,A -70.9232,B 24.8601,C -2.7293,E1 25.0692,E2 -205.8743} C_DIS
LIN {X 18.2744,Y -34.7877,Z 64,A -68.1966,B 24.8596,C -2.7337,E1 25.076,E2 -208.6039} C_DIS
LIN {X 19.9201,Y -33.8726,Z 64,A -65.1958,B 24.8587,C -2.7424,E1 25.0833,E2 -211.6164} C_DIS
LIN {X 21.987,Y -32.5689,Z 64,A -61.6857,B 24.8581,C -2.7484,E1 25.0915,E2 -215.1291} C_DIS
LIN {X 23.8246,Y -31.2503,Z 64,A -58.3194,B 24.8573,C -2.7562,E1 25.0991,E2 -218.5019} C_DIS
LIN {X 25.2709,Y -30.0926,Z 64,A -55.7765,B 24.857,C -2.7596,E1 25.1046,E2 -221.0431} C_DIS
LIN {X 26.8082,Y -28.7315,Z 64,A -52.8711,B 24.8564,C -2.765,E1 25.1106,E2 -223.9496} C_DIS
LIN {X 28.4416,Y -27.1149,Z 64,A -48.904,B 24.8545,C -2.7829,E1 25.1184,E2 -227.9422} C_DIS
LIN {X 30.4371,Y -24.8548,Z 64,A -44.9326,B 24.8541,C -2.7872,E1 25.1255,E2 -231.9056} C_DIS
LIN {X 31.7753,Y -23.1192,Z 64,A -41.8979,B 24.8535,C -2.793,E1 25.1306,E2 -234.9396} C_DIS
LIN {X 33.0267,Y -21.2931,Z 64,A -38.6781,B 24.8525,C -2.8017,E1 25.1356,E2 -238.1639} C_DIS
LIN {X 34.099,Y -19.5298,Z 64,A -35.4103,B 24.8512,C -2.8144,E1 25.1402,E2 -241.4451} C_DIS
LIN {X 35.2801,Y -17.3048,Z 64,A -32.4078,B 24.8512,C -2.814,E1 25.144,E2 -244.4308} C_DIS
LIN {X 36.3232,Y -14.9929,Z 64,A -28.62,B 24.8499,C -2.8264,E1 25.1483,E2 -248.2272} C_DIS
LIN {X 36.8088,Y -13.7581,Z 64,A -26.0914,B 24.8482,C -2.8421,E1 25.1508,E2 -250.7787} C_DIS
LIN {X 37.865,Y -10.5064,Z 64,A -20.9991,B 24.8464,C -2.8591,E1 25.1549,E2 -255.8824} C_DIS
LIN {X 38.577,Y -7.4813,Z 64,A -16.857,B 24.8456,C -2.8667,E1 25.1573,E2 -260.0184} C_DIS
LIN {X 39.0196,Y -4.6513,Z 64,A -12.5065,B 24.8439,C -2.8827,E1 25.159,E2 -264.3811} C_DIS
LIN {X 39.2625,Y -1.6177,Z 64,A -7.3716,B 24.8411,C -2.9084,E1 25.1598,E2 -269.5461} C_DIS
LIN {X 39.2407,Y 2.0814,Z 64,A -2.5788,B 24.8403,C -2.9151,E1 25.1593,E2 -274.3264} C_DIS
LIN {X 38.8823,Y 5.6862,Z 64,A 1.5732,B 24.8406,C -2.9127,E1 25.158,E2 -278.4482} C_DIS
LIN {X 38.5226,Y 7.7575,Z 64,A 5.9234,B 24.8372,C -2.9433,E1 25.1557,E2 -282.8453} C_DIS
LIN {X 37.7482,Y 10.9185,Z 64,A 10.2455,B 24.8364,C -2.9503,E1 25.1526,E2 -287.1593} C_DIS
LIN {X 36.914,Y 13.4722,Z 64,A 13.7228,B 24.836,C -2.9545,E1 25.1495,E2 -290.6268} C_DIS
LIN {X 36.1454,Y 15.4168,Z 64,A 17.3525,B 24.8339,C -2.9725,E1 25.1455,E2 -294.2792} C_DIS
LIN {X 34.6434,Y 18.5477,Z 64,A 22.0622,B 24.833,C -2.9805,E1 25.1396,E2 -298.9827} C_DIS
LIN {X 33.6648,Y 20.2696,Z 64,A 24.8144,B 24.8324,C -2.9858,E1 25.1357,E2 -301.7334} C_DIS
LIN {X 32.1976,Y 22.5274,Z 64,A 28.7362,B 24.8314,C -2.9955,E1 25.1296,E2 -305.6587} C_DIS
LIN {X 30.9469,Y 24.2173,Z 64,A 31.2957,B 24.8314,C -2.9948,E1 25.1253,E2 -308.2044} C_DIS
LIN {X 29.9405,Y 25.4501,Z 64,A 33.7488,B 24.8306,C -3.0022,E1 25.1209,E2 -310.6637} C_DIS
LIN {X 28.8753,Y 26.6525,Z 64,A 36.2755,B 24.8297,C -3.0102,E1 25.1162,E2 -313.1981} C_DIS
LIN {X 26.8779,Y 28.6659,Z 64,A 40.5437,B 24.8285,C -3.0207,E1 25.1077,E2 -317.4734} C_DIS
LIN {X 24.9469,Y 30.3618,Z 64,A 44.4149,B 24.8275,C -3.0296,E1 25.0994,E2 -321.3507} C_DIS
LIN {X 22.4637,Y 32.2419,Z 64,A 48.8238,B 24.8268,C -3.0353,E1 25.0895,E2 -325.7574} C_DIS
LIN {X 20.3797,Y 33.598,Z 64,A 52.5283,B 24.8261,C -3.0419,E1 25.0807,E2 -329.4657} C_DIS
LIN {X 18.2248,Y 34.8138,Z 64,A 55.5558,B 24.8265,C -3.0382,E1 25.0733,E2 -332.4756} C_DIS
LIN {X 16.2554,Y 35.7761,Z 64,A 59.4808,B 24.8249,C -3.0524,E1 25.0634,E2 -336.4245} C_DIS
LIN {X 13.8278,Y 36.7825,Z 64,A 63.0665,B 24.8249,C -3.0526,E1 25.0541,E2 -340.0026} C_DIS
LIN {X 11.0727,Y 37.7034,Z 64,A 67.3457,B 24.8244,C -3.0564,E1 25.0427,E2 -344.283} C_DIS
LIN {X 8.3277,Y 38.4032,Z 64,A 71.3439,B 24.8244,C -3.0568,E1 25.0318,E2 -348.2763} C_DIS
LIN {X 6.0061,Y 38.834,Z 64,A 74.6805,B 24.8244,C -3.0565,E1 25.0227,E2 -351.6088} C_DIS
LIN {X 4.0535,Y 39.086,Z 64,A 77.4451,B 24.8244,C -3.0556,E1 25.015,E2 -354.3691} C_DIS
LIN {X 2.0678,Y 39.2411,Z 64,A 80.8564,B 24.8237,C -3.0623,E1 25.0055,E2 -357.7951} C_DIS
LIN {X -0.7485,Y 39.2886,Z 64,A 84.703,B 24.8242,C -3.0581,E1 24.9947,E2 -361.6315} C_DIS
LIN {X -2.8135,Y 39.1951,Z 64,A 87.4977,B 24.8247,C -3.0541,E1 24.987,E2 -364.4176} C_DIS
LIN {X -6.187,Y 38.806,Z 64,A 92.1453,B 24.8254,C -3.0474,E1 24.9741,E2 -369.0524} C_DIS
LIN {X -8.2301,Y 38.4244,Z 64,A 96.1805,B 24.8243,C -3.0575,E1 24.963,E2 -373.1164} C_DIS
LIN {X -11.1897,Y 37.6689,Z 64,A 100.1829,B 24.8254,C -3.0474,E1 24.9523,E2 -377.1008} C_DIS
LIN {X -12.7133,Y 37.1825,Z 64,A 102.6777,B 24.8255,C -3.0466,E1 24.9457,E2 -379.5985} C_DIS
LIN {X -15.2189,Y 36.229,Z 64,A 106.1336,B 24.8267,C -3.036,E1 24.9368,E2 -383.0366} C_DIS
LIN {X -17.5636,Y 35.1524,Z 64,A 110.6999,B 24.8263,C -3.0397,E1 24.9252,E2 -387.6235} C_DIS
LIN {X -19.9489,Y 33.8556,Z 64,A 114.2127,B 24.8277,C -3.0277,E1 24.9167,E2 -391.118} C_DIS
LIN {X -22.0669,Y 32.5146,Z 64,A 117.8166,B 24.8285,C -3.0203,E1 24.9083,E2 -394.7159} C_DIS
LIN {X -24.2838,Y 30.8943,Z 64,A 122.2418,B 24.8289,C -3.0168,E1 24.8985,E2 -399.1487} C_DIS
LIN {X -26.1668,Y 29.3165,Z 64,A 125.1563,B 24.8307,C -3.0015,E1 24.8924,E2 -402.0383} C_DIS
LIN {X -28.002,Y 27.569,Z 64,A 129.6121,B 24.8307,C -3.0013,E1 24.8835,E2 -406.512} C_DIS
LIN {X -29.758,Y 25.6641,Z 64,A 132.7915,B 24.8325,C -2.9854,E1 24.8776,E2 -409.6678} C_DIS
LIN {X -31.2822,Y 23.7824,Z 64,A 136.7604,B 24.833,C -2.981,E1 24.8708,E2 -413.6448} C_DIS
LIN {X -32.9143,Y 21.4663,Z 64,A 141.0012,B 24.8341,C -2.971,E1 24.8641,E2 -417.8829} C_DIS
LIN {X -34.2067,Y 19.3417,Z 64,A 143.995,B 24.836,C -2.9542,E1 24.8599,E2 -420.852} C_DIS
LIN {X -35.1098,Y 17.6481,Z 64,A 147.2108,B 24.8364,C -2.9505,E1 24.8558,E2 -424.0761} C_DIS
LIN {X -35.9142,Y 15.9471,Z 64,A 149.9449,B 24.8373,C -2.9424,E1 24.8526,E2 -426.8057} C_DIS
LIN {X -36.5334,Y 14.4726,Z 64,A 152.3985,B 24.8379,C -2.9367,E1 24.8501,E2 -429.2594} C_DIS
LIN {X -37.3765,Y 12.1302,Z 64,A 155.9225,B 24.8393,C -2.9246,E1 24.8469,E2 -432.7745} C_DIS
LIN {X -38.1453,Y 9.4399,Z 64,A 159.5467,B 24.8412,C -2.9075,E1 24.8443,E2 -436.3787} C_DIS
LIN {X -38.5544,Y 7.5986,Z 64,A 163.1725,B 24.8412,C -2.9078,E1 24.8422,E2 -440.0268} C_DIS
LIN {X -39.0287,Y 4.5735,Z 64,A 167.6643,B 24.8426,C -2.8941,E1 24.8405,E2 -444.5126} C_DIS
LIN {X -39.2554,Y 1.7797,Z 64,A 171.451,B 24.8443,C -2.8782,E1 24.8398,E2 -448.2841} C_DIS
LIN {X -39.2942,Y -0.4001,Z 64,A 174.6961,B 24.8454,C -2.869,E1 24.8398,E2 -451.5265} C_DIS
LIN {X -39.2392,Y -2.1076,Z 64,A 177.1597,B 24.8462,C -2.8609,E1 24.8402,E2 -453.9857} C_DIS
LIN {X -39.0766,Y -4.144,Z 64,A 179.9599,B 24.8474,C -2.8499,E1 24.8409,E2 -456.7763} C_DIS
LIN {X -38.7641,Y -6.4421,Z 64,A -176.461,B 24.8483,C -2.8415,E1 24.8424,E2 -460.3568} C_DIS
LIN {X -38.3012,Y -8.7851,Z 64,A -172.9959,B 24.8495,C -2.8309,E1 24.8444,E2 -463.8167} C_DIS
LIN {X -37.8524,Y -10.5518,Z 64,A -170.1348,B 24.8501,C -2.8251,E1 24.8465,E2 -466.6805} C_DIS
LIN {X -36.9936,Y -13.2515,Z 64,A -166.2316,B 24.8516,C -2.8107,E1 24.8499,E2 -470.5717} C_DIS
LIN {X -36.3229,Y -14.9935,Z 64,A -163.7035,B 24.8526,C -2.801,E1 24.8525,E2 -473.0906} C_DIS
LIN {X -35.6073,Y -16.6216,Z 64,A -160.7581,B 24.853,C -2.7976,E1 24.8559,E2 -476.044} C_DIS
LIN {X -34.7161,Y -18.4104,Z 64,A -157.7145,B 24.8537,C -2.7911,E1 24.8598,E2 -479.0884} C_DIS
LIN {X -33.2017,Y -21.0198,Z 64,A -153.461,B 24.855,C -2.7782,E1 24.866,E2 -483.333} C_DIS
LIN {X -31.9145,Y -22.9268,Z 64,A -150.1043,B 24.8559,C -2.7701,E1 24.8713,E2 -486.6867} C_DIS
LIN {X -30.5583,Y -24.7052,Z 64,A -146.8226,B 24.8566,C -2.7627,E1 24.877,E2 -489.9662} C_DIS
LIN {X -28.8988,Y -26.6274,Z 64,A -142.8805,B 24.8572,C -2.7573,E1 24.8843,E2 -493.9131} C_DIS
LIN {X -27.2221,Y -28.3393,Z 64,A -139.581,B 24.8582,C -2.7479,E1 24.8908,E2 -497.204} C_DIS
LIN {X -25.4785,Y -29.9165,Z 64,A -136.0901,B 24.8588,C -2.7421,E1 24.8981,E2 -500.695} C_DIS
LIN {X -23.5856,Y -31.4305,Z 64,A -132.574,B 24.8594,C -2.7357,E1 24.9059,E2 -504.2087} C_DIS
LIN {X -21.9849,Y -32.5703,Z 64,A -129.3924,B 24.8595,C -2.7349,E1 24.9132,E2 -507.3991} C_DIS
LIN {X -19.0018,Y -34.3963,Z 64,A -124.1958,B 24.8601,C -2.729,E1 24.9258,E2 -512.5972} C_DIS
LIN {X -16.7765,Y -35.5344,Z 64,A -120.8178,B 24.8609,C -2.7215,E1 24.9342,E2 -515.966} C_DIS
LIN {X -14.2268,Y -36.6302,Z 64,A -116.5916,B 24.8611,C -2.7198,E1 24.9451,E2 -520.1975} C_DIS
LIN {X -11.376,Y -37.6129,Z 64,A -112.469,B 24.8618,C -2.7129,E1 24.9561,E2 -524.3114} C_DIS
LIN {X -9.2072,Y -38.2018,Z 64,A -108.9797,B 24.8617,C -2.7139,E1 24.9655,E2 -527.808} C_DIS
LIN {X -7.0441,Y -38.6593,Z 64,A -106.1916,B 24.8624,C -2.7069,E1 24.9731,E2 -530.5827} C_DIS
LIN {X -5.0088,Y -38.9752,Z 64,A -102.5106,B 24.8615,C -2.7153,E1 24.9834,E2 -534.2865} C_DIS
LIN {X -2.033,Y -39.2433,Z 64,A -98.651,B 24.8622,C -2.7086,E1 24.9941,E2 -538.1316} C_DIS
LIN {X -0.0824,Y -39.296,Z 64,A -95.3973,B 24.8616,C -2.7148,E1 25.0032,E2 -541.4001} C_DIS
LIN {X -0.0824,Y -39.296,Z 64,A -95.3973,B 24.8616,C -2.7148,E1 25.0032,E2 -541.4001} C_DIS
Enddeposition()
LIN {X 0.2461,Y -38.353,Z 64,A -95.2,B 24.8603,C -2.727,E1 25.0038,E2 -541.6264} C_DIS
Startdeposition()
$VEL.CP = VEL_PRINT
LIN {X -1.1221,Y -38.3406,Z 64,A -99.0061,B 24.8628,C -2.7033,E1 24.9931,E2 -537.7638} C_DIS
LIN {X -3.3931,Y -38.2066,Z 64,A -102.5037,B 24.8628,C -2.7021,E1 24.9833,E2 -534.2619} C_DIS
LIN {X -5.5638,Y -37.9511,Z 64,A -106.1073,B 24.8632,C -2.6985,E1 24.9733,E2 -530.647} C_DIS
LIN {X -7.8441,Y -37.5466,Z 64,A -109.1422,B 24.8626,C -2.7051,E1 24.965,E2 -527.6242} C_DIS
LIN {X -10.0764,Y -37.0099,Z 64,A -112.4656,B 24.8623,C -2.7083,E1 24.956,E2 -524.3037} C_DIS
LIN {X -12.3394,Y -36.3177,Z 64,A -115.7582,B 24.8617,C -2.7138,E1 24.9473,E2 -521.0184} C_DIS
LIN {X -14.3533,Y -35.5702,Z 64,A -119.5175,B 24.8621,C -2.7102,E1 24.9375,E2 -517.2425} C_DIS
LIN {X -16.8538,Y -34.4558,Z 64,A -123.4877,B 24.8614,C -2.7162,E1 24.9274,E2 -513.2766} C_DIS
LIN {X -18.7743,Y -33.4484,Z 64,A -126.4368,B 24.8607,C -2.7237,E1 24.9202,E2 -510.3372} C_DIS
LIN {X -20.5364,Y -32.3967,Z 64,A -129.7303,B 24.8605,C -2.7256,E1 24.9124,E2 -507.0378} C_DIS
LIN {X -22.3982,Y -31.1385,Z 64,A -133.0296,B 24.8599,C -2.7316,E1 24.9048,E2 -503.7417} C_DIS
LIN {X -24.2647,Y -29.707,Z 64,A -136.6449,B 24.8593,C -2.7367,E1 24.8969,E2 -500.1251} C_DIS
LIN {X -26.1011,Y -28.1076,Z 64,A -140.953,B 24.8593,C -2.7367,E1 24.888,E2 -495.7994} C_DIS
LIN {X -28.2241,Y -25.9743,Z 64,A -144.7108,B 24.8576,C -2.7539,E1 24.8808,E2 -492.0667} C_DIS
LIN {X -30.0472,Y -23.8418,Z 64,A -148.637,B 24.8563,C -2.7662,E1 24.8738,E2 -488.1516} C_DIS
LIN {X -31.1947,Y -22.3194,Z 64,A -151.829,B 24.8559,C -2.7694,E1 24.8685,E2 -484.952} C_DIS
LIN {X -32.487,Y -20.3927,Z 64,A -155.4279,B 24.8552,C -2.7767,E1 24.863,E2 -481.3525} C_DIS
LIN {X -33.5866,Y -18.5259,Z 64,A -158.4085,B 24.854,C -2.7878,E1 24.8589,E2 -478.3827} C_DIS
LIN {X -34.4032,Y -16.9608,Z 64,A -161.2235,B 24.8535,C -2.7931,E1 24.8554,E2 -475.5653} C_DIS
LIN {X -35.4241,Y -14.7112,Z 64,A -164.5518,B 24.852,C -2.8069,E1 24.8516,E2 -472.2519} C_DIS
LIN {X -36.0596,Y -13.0757,Z 64,A -168.1411,B 24.8522,C -2.805,E1 24.8481,E2 -468.6376} C_DIS
LIN {X -37.0696,Y -9.8537,Z 64,A -172.7126,B 24.8501,C -2.8244,E1 24.8446,E2 -464.0862} C_DIS
LIN {X -37.5657,Y -7.7512,Z 64,A -175.7488,B 24.8489,C -2.8359,E1 24.8427,E2 -461.0597} C_DIS
LIN {X -37.939,Y -5.6513,Z 64,A -179.5531,B 24.8485,C -2.8398,E1 24.841,E2 -457.2419} C_DIS
LIN {X -38.2691,Y -2.5955,Z 64,A 176.4063,B 24.8464,C -2.8592,E1 24.84,E2 -453.2236} C_DIS
LIN {X -38.3554,Y -0.4159,Z 64,A 173.0907,B 24.8454,C -2.8688,E1 24.8398,E2 -449.9111} C_DIS
LIN {X -38.3165,Y 1.7619,Z 64,A 169.6527,B 24.8445,C -2.8773,E1 24.8401,E2 -446.4726} C_DIS
LIN {X -38.1358,Y 4.1126,Z 64,A 165.5282,B 24.8439,C -2.8827,E1 24.8412,E2 -442.3363} C_DIS
LIN {X -37.6576,Y 7.2918,Z 64,A 161.4358,B 24.8415,C -2.9043,E1 24.8431,E2 -438.2714} C_DIS
LIN {X -37.2608,Y 9.1047,Z 64,A 158.0166,B 24.8412,C -2.9068,E1 24.8453,E2 -434.8381} C_DIS
LIN {X -36.3227,Y 12.3252,Z 64,A 153.7624,B 24.8388,C -2.9293,E1 24.8488,E2 -430.6132} C_DIS
LIN {X -35.7935,Y 13.7878,Z 64,A 151.2636,B 24.8382,C -2.9346,E1 24.8512,E2 -428.1129} C_DIS
LIN {X -35.1113,Y 15.4417,Z 64,A 148.0681,B 24.8379,C -2.9374,E1 24.8548,E2 -424.9066} C_DIS
LIN {X -33.5324,Y 18.6239,Z 64,A 142.1518,B 24.8368,C -2.9468,E1 24.8625,E2 -418.9813} C_DIS
LIN {X -31.1269,Y 22.4142,Z 64,A 136.5592,B 24.8336,C -2.9759,E1 24.8711,E2 -413.4304} C_DIS
LIN {X -30.1184,Y 23.7517,Z 64,A 133.5167,B 24.8334,C -2.977,E1 24.8763,E2 -410.3761} C_DIS
LIN {X -28.1149,Y 26.0925,Z 64,A 129.2151,B 24.8318,C -2.9914,E1 24.8843,E2 -406.0896} C_DIS
LIN {X -26.5527,Y 27.6806,Z 64,A 125.6313,B 24.8312,C -2.9965,E1 24.8914,E2 -402.5031} C_DIS
LIN {X -24.3726,Y 29.6188,Z 64,A 121.5809,B 24.8298,C -3.0092,E1 24.9,E2 -398.4673} C_DIS
LIN {X -22.8446,Y 30.8123,Z 64,A 118.0348,B 24.8298,C -3.0083,E1 24.9079,E2 -394.9063} C_DIS
LIN {X -19.5681,Y 32.9902,Z 64,A 113.2595,B 24.8273,C -3.0311,E1 24.919,E2 -390.17} C_DIS
LIN {X -17.9347,Y 33.9054,Z 64,A 109.3989,B 24.8281,C -3.0241,E1 24.9285,E2 -386.2818} C_DIS
LIN {X -14.8033,Y 35.3855,Z 64,A 104.8789,B 24.8264,C -3.039,E1 24.94,E2 -381.7861} C_DIS
LIN {X -13.1237,Y 36.0421,Z 64,A 102.3906,B 24.8257,C -3.0448,E1 24.9464,E2 -379.3065} C_DIS
LIN {X -11.5316,Y 36.5824,Z 64,A 99.4347,B 24.826,C -3.0426,E1 24.9543,E2 -376.34} C_DIS
LIN {X -9.3391,Y 37.203,Z 64,A 95.8491,B 24.8258,C -3.0438,E1 24.964,E2 -372.752} C_DIS
LIN {X -6.8492,Y 37.7406,Z 64,A 92.6873,B 24.8246,C -3.0545,E1 24.9726,E2 -369.6121} C_DIS
LIN {X -4.029,Y 38.1449,Z 64,A 88.5112,B 24.8242,C -3.0581,E1 24.9841,E2 -365.4412} C_DIS
LIN {X -2.4936,Y 38.2759,Z 64,A 85.6696,B 24.8248,C -3.0525,E1 24.9921,E2 -362.5851} C_DIS
LIN {X -0.2344,Y 38.3563,Z 64,A 82.3497,B 24.8247,C -3.0541,E1 25.0013,E2 -359.2687} C_DIS
LIN {X 2.5871,Y 38.2696,Z 64,A 78.2578,B 24.8244,C -3.0559,E1 25.0127,E2 -355.1823} C_DIS
LIN {X 4.7466,Y 38.0626,Z 64,A 74.7523,B 24.8249,C -3.0521,E1 25.0225,E2 -351.67} C_DIS
LIN {X 6.9787,Y 37.7173,Z 64,A 71.4357,B 24.8249,C -3.0517,E1 25.0316,E2 -348.356} C_DIS
LIN {X 9.3008,Y 37.2121,Z 64,A 68.1328,B 24.8248,C -3.0531,E1 25.0406,E2 -345.061} C_DIS
LIN {X 11.2543,Y 36.6688,Z 64,A 64.7403,B 24.8256,C -3.0462,E1 25.0497,E2 -341.6578} C_DIS
LIN {X 13.0075,Y 36.0841,Z 64,A 62.1014,B 24.8256,C -3.0455,E1 25.0566,E2 -339.0226} C_DIS
LIN {X 15.271,Y 35.1861,Z 64,A 58.3669,B 24.8262,C -3.0404,E1 25.0663,E2 -335.2847} C_DIS
LIN {X 17.1295,Y 34.3197,Z 64,A 55.4934,B 24.8263,C -3.0394,E1 25.0735,E2 -332.4164} C_DIS
LIN {X 18.8589,Y 33.4011,Z 64,A 52.5275,B 24.8269,C -3.0349,E1 25.0808,E2 -329.4484} C_DIS
LIN {X 20.7917,Y 32.2331,Z 64,A 49.1067,B 24.8275,C -3.0292,E1 25.0889,E2 -326.025} C_DIS
LIN {X 22.8046,Y 30.8422,Z 64,A 44.796,B 24.8293,C -3.0138,E1 25.0987,E2 -321.6928} C_DIS
LIN {X 25.1549,Y 28.9569,Z 64,A 40.9707,B 24.8291,C -3.0152,E1 25.1068,E2 -317.8856} C_DIS
LIN {X 27.1433,Y 27.102,Z 64,A 37.2995,B 24.8294,C -3.0127,E1 25.1142,E2 -314.2238} C_DIS
LIN {X 28.106,Y 26.1023,Z 64,A 35.2764,B 24.8298,C -3.009,E1 25.1181,E2 -312.2007} C_DIS
LIN {X 29.1543,Y 24.9257,Z 64,A 32.66,B 24.8309,C -2.9999,E1 25.1229,E2 -309.5744} C_DIS
LIN {X 30.5279,Y 23.224,Z 64,A 29.2939,B 24.8319,C -2.9907,E1 25.1287,E2 -306.2024} C_DIS
LIN {X 31.8713,Y 21.3429,Z 64,A 25.8624,B 24.8328,C -2.9825,E1 25.1342,E2 -302.7684} C_DIS
LIN {X 33.1838,Y 19.2382,Z 64,A 22.2169,B 24.8338,C -2.9739,E1 25.1394,E2 -299.1211} C_DIS
LIN {X 34.1952,Y 17.3762,Z 64,A 19.0635,B 24.8347,C -2.9656,E1 25.1435,E2 -295.9647} C_DIS
LIN {X 35.1982,Y 15.2433,Z 64,A 15.3786,B 24.8361,C -2.9533,E1 25.1478,E2 -292.2707} C_DIS
LIN {X 36.1775,Y 12.7456,Z 64,A 11.9703,B 24.8363,C -2.9512,E1 25.1511,E2 -288.8765} C_DIS
LIN {X 36.6497,Y 11.3164,Z 64,A 9.2976,B 24.8378,C -2.938,E1 25.1534,E2 -286.1875} C_DIS
LIN {X 37.2886,Y 8.9898,Z 64,A 5.4511,B 24.8394,C -2.9234,E1 25.1561,E2 -282.3288} C_DIS
LIN {X 37.8356,Y 6.3027,Z 64,A 1.9188,B 24.8398,C -2.9199,E1 25.1579,E2 -278.8088} C_DIS
LIN {X 38.0833,Y 4.5749,Z 64,A -0.7729,B 24.8408,C -2.9105,E1 25.1589,E2 -276.1108} C_DIS
LIN {X 38.2771,Y 2.4742,Z 64,A -4.0063,B 24.842,C -2.8994,E1 25.1596,E2 -272.8703} C_DIS
LIN {X 38.3582,Y 0.0292,Z 64,A -8.204,B 24.8442,C -2.8793,E1 25.1597,E2 -268.65} C_DIS
LIN {X 38.2559,Y -2.7831,Z 64,A -11.8541,B 24.8447,C -2.8749,E1 25.1592,E2 -265.0112} C_DIS
LIN {X 38.0867,Y -4.5465,Z 64,A -14.7003,B 24.8459,C -2.8635,E1 25.1583,E2 -262.1546} C_DIS
LIN {X 37.7188,Y -6.9685,Z 64,A -17.9288,B 24.8464,C -2.8589,E1 25.1568,E2 -258.9343} C_DIS
LIN {X 37.2944,Y -8.9655,Z 64,A -20.5092,B 24.8467,C -2.8569,E1 25.1552,E2 -256.3642} C_DIS
LIN {X 36.8861,Y -10.5207,Z 64,A -23.5287,B 24.8485,C -2.8396,E1 25.153,E2 -253.3212} C_DIS
LIN {X 36.0131,Y -13.203,Z 64,A -27.5803,B 24.8496,C -2.8294,E1 25.1494,E2 -249.2682} C_DIS
LIN {X 35.2796,Y -15.0539,Z 64,A -30.7832,B 24.8509,C -2.8169,E1 25.1459,E2 -246.0534} C_DIS
LIN {X 34.3069,Y -17.1556,Z 64,A -34.1488,B 24.8518,C -2.8083,E1 25.1418,E2 -242.6854} C_DIS
LIN {X 32.9734,Y -19.5964,Z 64,A -38.122,B 24.8528,C -2.7994,E1 25.1364,E2 -238.7117} C_DIS
LIN {X 31.7628,Y -21.5032,Z 64,A -41.1234,B 24.8532,C -2.7959,E1 25.1318,E2 -235.7171} C_DIS
LIN {X 30.7723,Y -22.8988,Z 64,A -44.0606,B 24.8545,C -2.7831,E1 25.127,E2 -232.764} C_DIS
LIN {X 29.4426,Y -24.5847,Z 64,A -47.3398,B 24.8555,C -2.7738,E1 25.1212,E2 -229.4778} C_DIS
LIN {X 27.7162,Y -26.5156,Z 64,A -50.9706,B 24.8561,C -2.7679,E1 25.1143,E2 -225.8491} C_DIS
LIN {X 26.4234,Y -27.8036,Z 64,A -53.8361,B 24.857,C -2.7594,E1 25.1086,E2 -222.9753} C_DIS
LIN {X 25.1276,Y -28.9807,Z 64,A -56.4801,B 24.8576,C -2.7531,E1 25.103,E2 -220.3269} C_DIS
LIN {X 23.2629,Y -30.4981,Z 64,A -60.0108,B 24.8583,C -2.7464,E1 25.0953,E2 -216.7934} C_DIS
LIN {X 21.472,Y -31.7839,Z 64,A -63.3503,B 24.8591,C -2.7392,E1 25.0876,E2 -213.4483} C_DIS
LIN {X 19.2427,Y -33.1813,Z 64,A -67.0865,B 24.8595,C -2.7349,E1 25.0787,E2 -209.7136} C_DIS
LIN {X 17.2544,Y -34.2571,Z 64,A -70.4283,B 24.86,C -2.7298,E1 25.0705,E2 -206.3691} C_DIS
LIN {X 14.5414,Y -35.4939,Z 64,A -75.6389,B 24.8618,C -2.7125,E1 25.057,E2 -201.1302} C_DIS
LIN {X 11.5549,Y -36.575,Z 64,A -79.2973,B 24.8609,C -2.7219,E1 25.0475,E2 -197.5013} C_DIS
LIN {X 9.9266,Y -37.0503,Z 64,A -82.3154,B 24.8618,C -2.7125,E1 25.0393,E2 -194.4657} C_DIS
LIN {X 7.5682,Y -37.6032,Z 64,A -86.397,B 24.8628,C -2.703,E1 25.0281,E2 -190.3668} C_DIS
LIN {X 4.1449,Y -38.1323,Z 64,A -90.9508,B 24.8623,C -2.708,E1 25.0156,E2 -185.8287} C_DIS
LIN {X 1.6254,Y -38.3226,Z 64,A -95.138,B 24.863,C -2.701,E1 25.0038,E2 -181.6264} C_DIS
LIN {X 1.6254,Y -38.3226,Z 64,A -95.138,B 24.863,C -2.701,E1 25.0038,E2 -181.6264} C_DIS
Enddeposition()
LIN {X 0.2408,Y -37.4136,Z 64,A -96.1482,B 24.86,C -2.7306,E1 25.0012,E2 -180.6869} C_DIS
Startdeposition()
$VEL.CP = VEL_PRINT
LIN {X 1.6554,Y -37.3817,Z 64,A -92.7169,B 24.8582,C -2.7479,E1 25.0109,E2 -184.1583} C_DIS
LIN {X 4.3321,Y -37.1667,Z 64,A -89.3765,B 24.859,C -2.7397,E1 25.0201,E2 -187.4773} C_DIS
LIN {X 5.7854,Y -36.9684,Z 64,A -86.7395,B 24.8583,C -2.7465,E1 25.0274,E2 -190.1281} C_DIS
LIN {X 7.8608,Y -36.5835,Z 64,A -83.6246,B 24.8583,C -2.7476,E1 25.036,E2 -193.2419} C_DIS
LIN {X 9.7567,Y -36.1239,Z 64,A -80.6788,B 24.858,C -2.75,E1 25.0439,E2 -196.189} C_DIS
LIN {X 11.8249,Y -35.501,Z 64,A -77.1845,B 24.8573,C -2.7565,E1 25.0533,E2 -199.6922} C_DIS
LIN {X 13.5305,Y -34.8867,Z 64,A -74.256,B 24.8567,C -2.7624,E1 25.0609,E2 -202.6282} C_DIS
LIN {X 16.2745,Y -33.6939,Z 64,A -69.9602,B 24.8564,C -2.7652,E1 25.0718,E2 -206.9198} C_DIS
LIN {X 17.8092,Y -32.9084,Z 64,A -67.0935,B 24.8556,C -2.7729,E1 25.0789,E2 -209.7967} C_DIS
LIN {X 19.9098,Y -31.6819,Z 64,A -63.6376,B 24.8553,C -2.7757,E1 25.0872,E2 -213.2485} C_DIS
LIN {X 21.6974,Y -30.4853,Z 64,A -60.3356,B 24.8546,C -2.7823,E1 25.0948,E2 -216.555} C_DIS
LIN {X 23.4239,Y -29.1802,Z 64,A -56.9006,B 24.8537,C -2.7911,E1 25.1023,E2 -219.9981} C_DIS
LIN {X 25.1994,Y -27.6611,Z 64,A -53.5398,B 24.8532,C -2.7958,E1 25.1094,E2 -223.3568} C_DIS
LIN {X 26.6657,Y -26.2503,Z 64,A -50.2743,B 24.8521,C -2.8055,E1 25.1159,E2 -226.6314} C_DIS
LIN {X 28.2105,Y -24.5825,Z 64,A -46.9374,B 24.8515,C -2.8119,E1 25.1221,E2 -229.9687} C_DIS
LIN {X 29.5835,Y -22.9118,Z 64,A -43.6252,B 24.8506,C -2.8205,E1 25.1279,E2 -233.2857} C_DIS
LIN {X 30.8797,Y -21.133,Z 64,A -40.1317,B 24.8494,C -2.8315,E1 25.1335,E2 -236.7882} C_DIS
LIN {X 32.3578,Y -18.7916,Z 64,A -36.0073,B 24.8483,C -2.8415,E1 25.1395,E2 -240.9153} C_DIS
LIN {X 33.4487,Y -16.773,Z 64,A -32.4925,B 24.8472,C -2.8517,E1 25.144,E2 -244.4355} C_DIS
LIN {X 34.2294,Y -15.1153,Z 64,A -29.0647,B 24.8453,C -2.8698,E1 25.1479,E2 -247.8878} C_DIS
LIN {X 35.3807,Y -12.1804,Z 64,A -24.9272,B 24.8449,C -2.8734,E1 25.1519,E2 -252.0104} C_DIS
LIN {X 36.0599,Y -9.99,Z 64,A -21.4277,B 24.8437,C -2.884,E1 25.1547,E2 -255.515} C_DIS
LIN {X 36.6056,Y -7.7573,Z 64,A -18.4008,B 24.8434,C -2.887,E1 25.1566,E2 -258.5316} C_DIS
LIN {X 36.9065,Y -6.1676,Z 64,A -15.3005,B 24.8415,C -2.9047,E1 25.1581,E2 -261.6556} C_DIS
LIN {X 37.2393,Y -3.6549,Z 64,A -12.0996,B 24.8413,C -2.906,E1 25.1591,E2 -264.8407} C_DIS
LIN {X 37.3637,Y -2.0209,Z 64,A -9.1417,B 24.8397,C -2.9211,E1 25.1597,E2 -267.8166} C_DIS
LIN {X 37.4189,Y 0.1105,Z 64,A -5.8123,B 24.8384,C -2.9323,E1 25.1597,E2 -271.1529} C_DIS
LIN {X 37.3481,Y 2.2965,Z 64,A -2.6981,B 24.8377,C -2.939,E1 25.1593,E2 -274.2644} C_DIS
LIN {X 37.1541,Y 4.4394,Z 64,A 0.4802,B 24.8367,C -2.9474,E1 25.1584,E2 -277.4437} C_DIS
LIN {X 36.8126,Y 6.7059,Z 64,A 4.3925,B 24.8348,C -2.9645,E1 25.1566,E2 -281.3735} C_DIS
LIN {X 36.2638,Y 9.2237,Z 64,A 7.9814,B 24.8341,C -2.9707,E1 25.1543,E2 -284.9563} C_DIS
LIN {X 35.7347,Y 11.0978,Z 64,A 10.9138,B 24.8332,C -2.9787,E1 25.152,E2 -287.891} C_DIS
LIN {X 35.0382,Y 13.1328,Z 64,A 13.7424,B 24.833,C -2.9809,E1 25.1494,E2 -290.7089} C_DIS
LIN {X 34.2498,Y 15.0695,Z 64,A 17.1281,B 24.8317,C -2.9928,E1 25.1457,E2 -294.1041} C_DIS
LIN {X 33.7382,Y 16.1817,Z 64,A 19.9782,B 24.8294,C -3.0131,E1 25.1423,E2 -296.9869} C_DIS
LIN {X 32.3111,Y 18.8722,Z 64,A 24.0648,B 24.829,C -3.0164,E1 25.1367,E2 -301.0602} C_DIS
LIN {X 31.1858,Y 20.6781,Z 64,A 27.1096,B 24.8284,C -3.0214,E1 25.1321,E2 -304.1015} C_DIS
LIN {X 30.0697,Y 22.2705,Z 64,A 30.236,B 24.8273,C -3.0308,E1 25.127,E2 -307.2351} C_DIS
LIN {X 28.6722,Y 24.0429,Z 64,A 33.6049,B 24.8266,C -3.0375,E1 25.121,E2 -310.6041} C_DIS
LIN {X 27.1974,Y 25.699,Z 64,A 36.8415,B 24.826,C -3.0425,E1 25.115,E2 -313.8384} C_DIS
LIN {X 26.0721,Y 26.8402,Z 64,A 39.5021,B 24.8251,C -3.0506,E1 25.1096,E2 -316.5069} C_DIS
LIN {X 24.4711,Y 28.3077,Z 64,A 42.4477,B 24.825,C -3.0515,E1 25.1035,E2 -319.4429} C_DIS
LIN {X 22.9204,Y 29.5769,Z 64,A 45.7448,B 24.8239,C -3.0603,E1 25.0963,E2 -322.7485} C_DIS
LIN {X 21.29,Y 30.7713,Z 64,A 48.8246,B 24.8234,C -3.0652,E1 25.0893,E2 -325.8293} C_DIS
LIN {X 19.5708,Y 31.8926,Z 64,A 51.9727,B 24.8228,C -3.07,E1 25.0819,E2 -328.9787} C_DIS
LIN {X 17.7445,Y 32.9435,Z 64,A 55.2858,B 24.8222,C -3.0756,E1 25.0738,E2 -332.2953} C_DIS
LIN {X 16.1796,Y 33.7395,Z 64,A 57.5868,B 24.8224,C -3.0735,E1 25.0681,E2 -334.5852} C_DIS
LIN {X 13.4229,Y 34.9281,Z 64,A 62.1624,B 24.8219,C -3.0779,E1 25.0563,E2 -339.1605} C_DIS
LIN {X 10.8656,Y 35.8058,Z 64,A 67.2328,B 24.8201,C -3.0937,E1 25.0427,E2 -344.2588} C_DIS
LIN {X 7.8051,Y 36.5954,Z 64,A 71.4603,B 24.8207,C -3.0881,E1 25.0313,E2 -348.4672} C_DIS
LIN {X 5.676,Y 36.9853,Z 64,A 74.8064,B 24.8205,C -3.0896,E1 25.0221,E2 -351.8133} C_DIS
LIN {X 3.5141,Y 37.253,Z 64,A 77.7411,B 24.8211,C -3.085,E1 25.014,E2 -354.7351} C_DIS
LIN {X 1.9697,Y 37.3665,Z 64,A 80.5862,B 24.8204,C -3.091,E1 25.006,E2 -357.5932} C_DIS
LIN {X -0.3406,Y 37.4169,Z 64,A 84.0309,B 24.8206,C -3.0892,E1 24.9964,E2 -361.0334} C_DIS
LIN {X -2.5377,Y 37.3322,Z 64,A 87.4429,B 24.8206,C -3.0885,E1 24.9869,E2 -364.4448} C_DIS
LIN {X -4.7251,Y 37.1189,Z 64,A 90.415,B 24.8214,C -3.082,E1 24.9787,E2 -367.4032} C_DIS
LIN {X -6.581,Y 36.8351,Z 64,A 93.2897,B 24.8217,C -3.08,E1 24.9708,E2 -370.2758} C_DIS
LIN {X -8.3165,Y 36.4826,Z 64,A 96.3732,B 24.8214,C -3.0821,E1 24.9623,E2 -373.368} C_DIS
LIN {X -10.4359,Y 35.9334,Z 64,A 99.7252,B 24.8218,C -3.0787,E1 24.9533,E2 -376.717} C_DIS
LIN {X -12.5211,Y 35.2611,Z 64,A 103.0709,B 24.8223,C -3.0746,E1 24.9445,E2 -380.0593} C_DIS
LIN {X -14.3878,Y 34.542,Z 64,A 106.5201,B 24.8223,C -3.0748,E1 24.9355,E2 -383.5167} C_DIS
LIN {X -17.5575,Y 33.0437,Z 64,A 111.6276,B 24.8236,C -3.0635,E1 24.9228,E2 -388.6107} C_DIS
LIN {X -19.5546,Y 31.9025,Z 64,A 115.1001,B 24.8244,C -3.0567,E1 24.9145,E2 -392.0775} C_DIS
LIN {X -20.7775,Y 31.1202,Z 64,A 117.4212,B 24.8247,C -3.0536,E1 24.9091,E2 -394.3988} C_DIS
LIN {X -22.9098,Y 29.5851,Z 64,A 120.7707,B 24.8265,C -3.0384,E1 24.9016,E2 -397.7239} C_DIS
LIN {X -24.8207,Y 28.0017,Z 64,A 125.977,B 24.8257,C -3.0448,E1 24.8905,E2 -402.9656} C_DIS
LIN {X -27.011,Y 25.8949,Z 64,A 130.6882,B 24.8269,C -3.0343,E1 24.8813,E2 -407.672} C_DIS
LIN {X -30.0098,Y 22.351,Z 64,A 137.0849,B 24.8298,C -3.0089,E1 24.8701,E2 -414.0377} C_DIS
LIN {X -31.6025,Y 20.0359,Z 64,A 141.416,B 24.8311,C -2.9975,E1 24.8634,E2 -418.3632} C_DIS
LIN {X -32.7446,Y 18.109,Z 64,A 144.8097,B 24.8323,C -2.9875,E1 24.8587,E2 -421.7506} C_DIS
LIN {X -33.7569,Y 16.143,Z 64,A 147.9573,B 24.8336,C -2.9754,E1 24.8548,E2 -424.8862} C_DIS
LIN {X -34.611,Y 14.2202,Z 64,A 151.5344,B 24.8343,C -2.9693,E1 24.8509,E2 -428.4685} C_DIS
LIN {X -35.2608,Y 12.5217,Z 64,A 154.9216,B 24.8346,C -2.9668,E1 24.8477,E2 -431.8688} C_DIS
LIN {X -36.4298,Y 8.545,Z 64,A 160.6808,B 24.8374,C -2.9416,E1 24.8435,E2 -437.6012} C_DIS
LIN {X -36.8953,Y 6.2347,Z 64,A 164.2969,B 24.8386,C -2.9304,E1 24.8416,E2 -441.212} C_DIS
LIN {X -37.1972,Y 4.0609,Z 64,A 167.6822,B 24.8398,C -2.9202,E1 24.8405,E2 -444.5929} C_DIS
LIN {X -37.3734,Y 1.8328,Z 64,A 171.1622,B 24.8409,C -2.91,E1 24.8399,E2 -448.0695} C_DIS
LIN {X -37.4163,Y -0.4317,Z 64,A 174.68,B 24.842,C -2.8996,E1 24.8399,E2 -451.5836} C_DIS
LIN {X -37.3202,Y -2.7129,Z 64,A 178.1402,B 24.8432,C -2.8884,E1 24.8404,E2 -455.0378} C_DIS
LIN {X -37.1027,Y -4.8497,Z 64,A -178.5543,B 24.8443,C -2.8784,E1 24.8415,E2 -458.3392} C_DIS
LIN {X -36.7456,Y -7.0631,Z 64,A -175.0354,B 24.8454,C -2.8688,E1 24.8432,E2 -461.8559} C_DIS
LIN {X -36.282,Y -9.1514,Z 64,A -171.1632,B 24.8458,C -2.8648,E1 24.8457,E2 -465.7413} C_DIS
LIN {X -35.3818,Y -12.1769,Z 64,A -166.9296,B 24.848,C -2.8448,E1 24.8493,E2 -469.9513} C_DIS
LIN {X -34.6035,Y -14.2386,Z 64,A -163.4257,B 24.8488,C -2.8365,E1 24.8529,E2 -473.455} C_DIS
LIN {X -33.6617,Y -16.3414,Z 64,A -159.6729,B 24.8496,C -2.8291,E1 24.8574,E2 -477.2105} C_DIS
LIN {X -32.4434,Y -18.6427,Z 64,A -155.8015,B 24.8509,C -2.8174,E1 24.8626,E2 -481.0743} C_DIS
LIN {X -31.1733,Y -20.697,Z 64,A -152.2334,B 24.852,C -2.8068,E1 24.868,E2 -484.635} C_DIS
LIN {X -29.9029,Y -22.4933,Z 64,A -148.8553,B 24.8529,C -2.7988,E1 24.8735,E2 -488.0104} C_DIS
LIN {X -28.5735,Y -24.16,Z 64,A -145.7156,B 24.8538,C -2.7901,E1 24.8791,E2 -491.1437} C_DIS
LIN {X -27.2376,Y -25.6563,Z 64,A -142.2849,B 24.8541,C -2.7872,E1 24.8856,E2 -494.5828} C_DIS
LIN {X -25.4274,Y -27.452,Z 64,A -138.4402,B 24.855,C -2.7788,E1 24.8933,E2 -498.4232} C_DIS
LIN {X -23.6844,Y -28.9691,Z 64,A -134.8718,B 24.8556,C -2.7726,E1 24.901,E2 -501.9906} C_DIS
LIN {X -21.8098,Y -30.4051,Z 64,A -131.3792,B 24.8564,C -2.7651,E1 24.9088,E2 -505.4777} C_DIS
LIN {X -19.9687,Y -31.6451,Z 64,A -127.8299,B 24.8567,C -2.7616,E1 24.9171,E2 -509.0302} C_DIS
LIN {X -18.3816,Y -32.5925,Z 64,A -124.4024,B 24.8564,C -2.7647,E1 24.9255,E2 -512.4751} C_DIS
LIN {X -15.4724,Y -34.0697,Z 64,A -120.5561,B 24.8584,C -2.7455,E1 24.935,E2 -516.2856} C_DIS
LIN {X -13.4912,Y -34.9017,Z 64,A -116.4751,B 24.8578,C -2.7516,E1 24.9457,E2 -520.3902} C_DIS
LIN {X -10.8437,Y -35.8125,Z 64,A -112.537,B 24.8586,C -2.7442,E1 24.9561,E2 -524.3178} C_DIS
LIN {X -8.7555,Y -36.3794,Z 64,A -109.2645,B 24.8588,C -2.7419,E1 24.9649,E2 -527.5895} C_DIS
LIN {X -6.6608,Y -36.8207,Z 64,A -106.0577,B 24.859,C -2.7397,E1 24.9737,E2 -530.7948} C_DIS
LIN {X -4.7992,Y -37.1093,Z 64,A -102.8588,B 24.8587,C -2.7431,E1 24.9826,E2 -534.0042} C_DIS
LIN {X -2.423,Y -37.3398,Z 64,A -99.4248,B 24.859,C -2.7401,E1 24.9921,E2 -537.4327} C_DIS
LIN {X -0.3466,Y -37.4169,Z 64,A -96.1743,B 24.8588,C -2.7415,E1 25.0012,E2 -540.6869} C_DIS
LIN {X -0.3466,Y -37.4169,Z 64,A -96.1743,B 24.8588,C -2.7415,E1 25.0012,E2 -540.6869} C_DIS
Enddeposition()
LIN {X 0.2245,Y -36.4765,Z 64,A -95.5364,B 24.8575,C -2.7547,E1 25.0031,E2 -541.356} C_DIS
Startdeposition()
$VEL.CP = VEL_PRINT
LIN {X -0.8858,Y -36.4689,Z 64,A -98.5931,B 24.8592,C -2.7379,E1 24.9944,E2 -538.2592} C_DIS
LIN {X -2.6839,Y -36.3813,Z 64,A -101.7568,B 24.8596,C -2.7337,E1 24.9856,E2 -535.0845} C_DIS
LIN {X -5.1972,Y -36.1074,Z 64,A -104.641,B 24.8582,C -2.7474,E1 24.9777,E2 -532.231} C_DIS
LIN {X -7.11,Y -35.7803,Z 64,A -108.4213,B 24.859,C -2.7396,E1 24.9672,E2 -528.4285} C_DIS
LIN {X -8.8663,Y -35.386,Z 64,A -111.2893,B 24.859,C -2.7406,E1 24.9594,E2 -525.5589} C_DIS
LIN {X -10.928,Y -34.8042,Z 64,A -114.6944,B 24.8587,C -2.7424,E1 24.9503,E2 -522.1524} C_DIS
LIN {X -12.7273,Y -34.1878,Z 64,A -117.6591,B 24.8585,C -2.7451,E1 24.9425,E2 -519.1884} C_DIS
LIN {X -14.3798,Y -33.5261,Z 64,A -120.6377,B 24.8584,C -2.7459,E1 24.9348,E2 -516.2047} C_DIS
LIN {X -16.661,Y -32.4521,Z 64,A -123.6806,B 24.8569,C -2.7606,E1 24.9272,E2 -513.1891} C_DIS
LIN {X -18.6963,Y -31.3245,Z 64,A -127.1573,B 24.8562,C -2.7673,E1 24.9187,E2 -509.7185} C_DIS
LIN {X -20.2703,Y -30.3302,Z 64,A -131.0088,B 24.8567,C -2.7618,E1 24.9096,E2 -505.8414} C_DIS
LIN {X -21.6946,Y -29.3281,Z 64,A -133.9772,B 24.8565,C -2.7638,E1 24.9029,E2 -502.8676} C_DIS
LIN {X -23.4805,Y -27.9187,Z 64,A -137.5286,B 24.8558,C -2.7705,E1 24.8952,E2 -499.3187} C_DIS
LIN {X -25.1458,Y -26.4288,Z 64,A -141.0667,B 24.8551,C -2.7771,E1 24.8879,E2 -495.782} C_DIS
LIN {X -27.0194,Y -24.5102,Z 64,A -144.2207,B 24.8531,C -2.7966,E1 24.8819,E2 -492.6609} C_DIS
LIN {X -28.1992,Y -23.1432,Z 64,A -148.1498,B 24.8536,C -2.7921,E1 24.8747,E2 -488.7032} C_DIS
LIN {X -29.5672,Y -21.3679,Z 64,A -151.4953,B 24.8525,C -2.8022,E1 24.8691,E2 -485.3656} C_DIS
LIN {X -30.5717,Y -19.9037,Z 64,A -154.3016,B 24.8518,C -2.8089,E1 24.8648,E2 -482.5615} C_DIS
LIN {X -31.6462,Y -18.146,Z 64,A -156.9108,B 24.8503,C -2.8232,E1 24.8611,E2 -479.973} C_DIS
LIN {X -32.5838,Y -16.4031,Z 64,A -160.6858,B 24.8501,C -2.8252,E1 24.8561,E2 -476.1827} C_DIS
LIN {X -33.3519,Y -14.7785,Z 64,A -163.4841,B 24.8492,C -2.8332,E1 24.8528,E2 -473.3883} C_DIS
LIN {X -34.0312,Y -13.1402,Z 64,A -166.3533,B 24.8484,C -2.8403,E1 24.8499,E2 -470.52} C_DIS
LIN {X -34.6372,Y -11.4476,Z 64,A -169.1881,B 24.8476,C -2.8483,E1 24.8473,E2 -467.6883} C_DIS
LIN {X -35.1555,Y -9.7388,Z 64,A -172.179,B 24.8469,C -2.8549,E1 24.845,E2 -464.6959} C_DIS
LIN {X -35.6888,Y -7.5557,Z 64,A -175.5439,B 24.8456,C -2.867,E1 24.8429,E2 -461.3401} C_DIS
LIN {X -36.0145,Y -5.8099,Z 64,A -178.3581,B 24.8447,C -2.8752,E1 24.8415,E2 -458.529} C_DIS
LIN {X -36.2555,Y -4.0377,Z 64,A 178.8051,B 24.8438,C -2.8836,E1 24.8406,E2 -455.6954} C_DIS
LIN {X -36.4114,Y -2.2347,Z 64,A 175.9664,B 24.8428,C -2.8925,E1 24.84,E2 -452.8608} C_DIS
LIN {X -36.481,Y -0.0005,Z 64,A 172.0302,B 24.842,C -2.8997,E1 24.8398,E2 -448.9181} C_DIS
LIN {X -36.4123,Y 2.2216,Z 64,A 168.869,B 24.8405,C -2.9136,E1 24.8402,E2 -445.771} C_DIS
LIN {X -36.1868,Y 4.6103,Z 64,A 165.6906,B 24.8386,C -2.9306,E1 24.8411,E2 -442.6145} C_DIS
LIN {X -35.8245,Y 6.8821,Z 64,A 161.2964,B 24.8381,C -2.9349,E1 24.8431,E2 -438.2045} C_DIS
LIN {X -35.3458,Y 9.0244,Z 64,A 157.7176,B 24.8371,C -2.9444,E1 24.8455,E2 -434.6274} C_DIS
LIN {X -34.6353,Y 11.4537,Z 64,A 153.954,B 24.8355,C -2.9584,E1 24.8486,E2 -430.8757} C_DIS
LIN {X -34.0441,Y 13.1065,Z 64,A 151.1851,B 24.8346,C -2.9666,E1 24.8512,E2 -428.1107} C_DIS
LIN {X -33.3502,Y 14.7822,Z 64,A 148.3453,B 24.8337,C -2.9751,E1 24.8544,E2 -425.2756} C_DIS
LIN {X -32.5878,Y 16.3952,Z 64,A 145.5507,B 24.8327,C -2.9833,E1 24.8578,E2 -422.4854} C_DIS
LIN {X -31.7415,Y 17.9801,Z 64,A 142.6697,B 24.8319,C -2.9907,E1 24.8616,E2 -419.6071} C_DIS
LIN {X -30.8309,Y 19.4999,Z 64,A 139.8797,B 24.831,C -2.9984,E1 24.8657,E2 -416.8211} C_DIS
LIN {X -29.8414,Y 20.9828,Z 64,A 137.0684,B 24.8302,C -3.0058,E1 24.8701,E2 -414.0136} C_DIS
LIN {X -28.69,Y 22.5312,Z 64,A 133.8554,B 24.8295,C -3.012,E1 24.8756,E2 -410.8001} C_DIS
LIN {X -27.2975,Y 24.2001,Z 64,A 130.4054,B 24.8286,C -3.0202,E1 24.8819,E2 -407.354} C_DIS
LIN {X -25.8049,Y 25.7859,Z 64,A 127.0149,B 24.8276,C -3.0286,E1 24.8884,E2 -403.9691} C_DIS
LIN {X -24.288,Y 27.2188,Z 64,A 123.6937,B 24.8268,C -3.0356,E1 24.8953,E2 -400.6511} C_DIS
LIN {X -22.6023,Y 28.6337,Z 64,A 120.2188,B 24.826,C -3.0428,E1 24.9028,E2 -397.1803} C_DIS
LIN {X -21.0024,Y 29.8277,Z 64,A 117.2177,B 24.8251,C -3.0503,E1 24.9095,E2 -394.1868} C_DIS
LIN {X -19.3655,Y 30.9151,Z 64,A 113.9338,B 24.8247,C -3.0541,E1 24.9173,E2 -390.9012} C_DIS
LIN {X -17.6038,Y 31.9516,Z 64,A 110.8627,B 24.8239,C -3.061,E1 24.9247,E2 -387.8377} C_DIS
LIN {X -16.0102,Y 32.7785,Z 64,A 108.0784,B 24.8233,C -3.0658,E1 24.9316,E2 -385.0574} C_DIS
LIN {X -14.1067,Y 33.6418,Z 64,A 104.6626,B 24.8229,C -3.0691,E1 24.9404,E2 -381.6414} C_DIS
LIN {X -12.2986,Y 34.3438,Z 64,A 101.7314,B 24.8223,C -3.0743,E1 24.948,E2 -378.7163} C_DIS
LIN {X -10.6008,Y 34.9052,Z 64,A 98.8853,B 24.822,C -3.077,E1 24.9556,E2 -375.8718} C_DIS
LIN {X -8.8657,Y 35.3861,Z 64,A 96.0585,B 24.8217,C -3.0798,E1 24.9632,E2 -373.0475} C_DIS
LIN {X -7.114,Y 35.7795,Z 64,A 93.2494,B 24.8214,C -3.0823,E1 24.9709,E2 -370.2409} C_DIS
LIN {X -5.3451,Y 36.0863,Z 64,A 90.3991,B 24.8212,C -3.0839,E1 24.9787,E2 -367.3918} C_DIS
LIN {X -3.5831,Y 36.3031,Z 64,A 87.6461,B 24.821,C -3.0858,E1 24.9864,E2 -364.6416} C_DIS
LIN {X -1.7875,Y 36.4358,Z 64,A 84.7945,B 24.8209,C -3.0866,E1 24.9943,E2 -361.791} C_DIS
LIN {X -0.0122,Y 36.4802,Z 64,A 81.9583,B 24.8209,C -3.0866,E1 25.0022,E2 -358.9549} C_DIS
LIN {X 2.0922,Y 36.4192,Z 64,A 79.427,B 24.8198,C -3.0963,E1 25.0092,E2 -356.4471} C_DIS
LIN {X 4.0262,Y 36.2567,Z 64,A 75.9524,B 24.8204,C -3.0908,E1 25.0189,E2 -352.9614} C_DIS
LIN {X 5.7861,Y 36.0184,Z 64,A 72.8219,B 24.821,C -3.0859,E1 25.0276,E2 -349.8221} C_DIS
LIN {X 7.8879,Y 35.6168,Z 64,A 69.3909,B 24.8212,C -3.0836,E1 25.037,E2 -346.3897} C_DIS
LIN {X 9.7508,Y 35.1521,Z 64,A 66.4959,B 24.8212,C -3.0833,E1 25.0448,E2 -343.4985} C_DIS
LIN {X 11.453,Y 34.6355,Z 64,A 63.4317,B 24.8219,C -3.0777,E1 25.053,E2 -340.4267} C_DIS
LIN {X 13.543,Y 33.8723,Z 64,A 60.2187,B 24.8219,C -3.0781,E1 25.0613,E2 -337.2216} C_DIS
LIN {X 15.1889,Y 33.1673,Z 64,A 57.3785,B 24.8223,C -3.0746,E1 25.0686,E2 -334.3802} C_DIS
LIN {X 16.8061,Y 32.3779,Z 64,A 54.6049,B 24.8226,C -3.0719,E1 25.0755,E2 -331.6075} C_DIS
LIN {X 18.3722,Y 31.5161,Z 64,A 51.7734,B 24.8231,C -3.0677,E1 25.0824,E2 -328.7745} C_DIS
LIN {X 19.8834,Y 30.585,Z 64,A 49.0073,B 24.8235,C -3.0638,E1 25.0889,E2 -326.008} C_DIS
LIN {X 21.3677,Y 29.5673,Z 64,A 46.1986,B 24.824,C -3.0594,E1 25.0953,E2 -323.1986} C_DIS
LIN {X 22.7901,Y 28.4853,Z 64,A 43.1939,B 24.8249,C -3.0517,E1 25.1019,E2 -320.1868} C_DIS
LIN {X 24.4993,Y 27.0295,Z 64,A 39.6692,B 24.8257,C -3.045,E1 25.1093,E2 -316.66} C_DIS
LIN {X 26.3641,Y 25.2131,Z 64,A 36.5778,B 24.825,C -3.0507,E1 25.1154,E2 -313.5953} C_DIS
LIN {X 27.6266,Y 23.8235,Z 64,A 32.6854,B 24.8273,C -3.0307,E1 25.1227,E2 -309.6727} C_DIS
LIN {X 29.0292,Y 22.0932,Z 64,A 29.265,B 24.8282,C -3.0236,E1 25.1286,E2 -306.2516} C_DIS
LIN {X 30.3303,Y 20.2703,Z 64,A 25.883,B 24.8289,C -3.017,E1 25.134,E2 -302.8705} C_DIS
LIN {X 31.2799,Y 18.7714,Z 64,A 23.1312,B 24.8297,C -3.0104,E1 25.1381,E2 -300.117} C_DIS
LIN {X 32.3779,Y 16.8053,Z 64,A 20.0926,B 24.8299,C -3.0084,E1 25.1421,E2 -297.0896} C_DIS
LIN {X 33.2649,Y 14.9737,Z 64,A 16.2896,B 24.8319,C -2.9906,E1 25.1467,E2 -293.2649} C_DIS
LIN {X 34.0341,Y 13.1326,Z 64,A 13.2939,B 24.8327,C -2.9838,E1 25.1498,E2 -290.2696} C_DIS
LIN {X 34.6401,Y 11.4389,Z 64,A 10.4952,B 24.8336,C -2.976,E1 25.1524,E2 -287.4683} C_DIS
LIN {X 35.2111,Y 9.5365,Z 64,A 7.2322,B 24.8348,C -2.9646,E1 25.1549,E2 -284.197} C_DIS
LIN {X 35.6881,Y 7.5588,Z 64,A 4.2352,B 24.8356,C -2.958,E1 25.1567,E2 -281.2018} C_DIS
LIN {X 36.0166,Y 5.7975,Z 64,A 1.4317,B 24.8365,C -2.9496,E1 25.1581,E2 -278.3947} C_DIS
LIN {X 36.2566,Y 4.0276,Z 64,A -1.3397,B 24.8374,C -2.9415,E1 25.159,E2 -275.6205} C_DIS
LIN {X 36.4114,Y 2.2349,Z 64,A -4.1293,B 24.8383,C -2.9332,E1 25.1596,E2 -272.828} C_DIS
LIN {X 36.481,Y 0.0041,Z 64,A -7.6991,B 24.8396,C -2.9213,E1 25.1598,E2 -269.251} C_DIS
LIN {X 36.436,Y -1.7839,Z 64,A -10.3816,B 24.8404,C -2.9144,E1 25.1595,E2 -266.5683} C_DIS
LIN {X 36.3037,Y -3.5773,Z 64,A -13.1953,B 24.8414,C -2.9057,E1 25.1588,E2 -263.7507} C_DIS
LIN {X 36.0856,Y -5.3499,Z 64,A -16.0138,B 24.8423,C -2.8967,E1 25.1578,E2 -260.9275} C_DIS
LIN {X 35.78,Y -7.1114,Z 64,A -18.7951,B 24.8433,C -2.8883,E1 25.1563,E2 -258.1427} C_DIS
LIN {X 35.3861,Y -8.866,Z 64,A -21.6189,B 24.8442,C -2.8796,E1 25.1545,E2 -255.3146} C_DIS
LIN {X 34.9128,Y -10.5757,Z 64,A -24.3348,B 24.845,C -2.8721,E1 25.1524,E2 -252.5965} C_DIS
LIN {X 34.349,Y -12.2838,Z 64,A -27.1322,B 24.8459,C -2.864,E1 25.1499,E2 -249.7955} C_DIS
LIN {X 33.7122,Y -13.9379,Z 64,A -29.9512,B 24.8469,C -2.8551,E1 25.147,E2 -246.9712} C_DIS
Enddeposition()
END
